LIN {X 0,Y 520.73,Z 981.897,A -85,B 0,C 180,E1 23653.264,E2 23653.264} C_VEL
LIN {X 0,Y 521.246,Z 970.847,A -85,B 0,C 180,E1 23650.972,E2 23650.972} C_VEL
LIN {X 0,Y 521.946,Z 957.782,A -85,B 0,C 180,E1 23648.66,E2 23648.66} C_VEL
LIN {X 0,Y 522.858,Z 943.401,A -85,B 0,C 180,E1 23646.447,E2 23646.447} C_VEL
LIN {X 0,Y 523.895,Z 928.064,A -85,B 0,C 180,E1 23644.403,E2 23644.403} C_VEL
LIN {X 0,Y 525.181,Z 910.158,A -85,B 0,C 180,E1 23642.324,E2 23642.324} C_VEL
LIN {X 0,Y 526.584,Z 891.948,A -85,B 0,C 180,E1 23640.484,E2 23640.484} C_VEL
LIN {X 0,Y 527.978,Z 872.899,A -85,B 0,C 180,E1 23638.832,E2 23638.832} C_VEL
LIN {X 0,Y 529.539,Z 851.797,A -85,B 0,C 180,E1 23637.256,E2 23637.256} C_VEL
LIN {X 0,Y 530.892,Z 831.885,A -85,B 0,C 180,E1 23635.993,E2 23635.993} C_VEL
LIN {X 0,Y 532.275,Z 810.339,A -85,B 0,C 180,E1 23634.853,E2 23634.853} C_VEL
LIN {X 0,Y 533.339,Z 791.087,A -85,B 0,C 180,E1 23634.009,E2 23634.009} C_VEL
LIN {X 0,Y 534.431,Z 767.293,A -85,B 0,C 180,E1 23633.183,E2 23633.183} C_VEL
LIN {X 0,Y 535.229,Z 746.117,A -85,B 0,C 180,E1 23632.64,E2 23632.64} C_VEL
LIN {X 0,Y 535.849,Z 714.207,A -85,B 0,C 180,E1 23632.087,E2 23632.087} C_VEL
LIN {X 0,Y 538.701,Z 503.345,A -85,B 0,C 180,E1 23628.756,E2 23628.756} C_VEL
LIN {X 0,Y 539.867,Z 409.94,A -85,B 0,C 180,E1 23627.231,E2 23627.231} C_VEL
LIN {X 0,Y 537.549,Z 399.203,A -85,B 0,C 180,E1 23626.813,E2 23626.813} C_VEL
LIN {X 0,Y 531.853,Z 390.282,A -85,B 0,C 180,E1 23626.056,E2 23626.056} C_VEL
LIN {X 0,Y 523.904,Z 373.802,A -85,B 0,C 180,E1 23623.836,E2 23623.836} C_VEL
LIN {X 0,Y 520.61,Z 366.663,A -85,B 0,C 180,E1 23622.813,E2 23622.813} C_VEL
LIN {X 0,Y 520.571,Z 366.179,A -85,B 0,C 180,E1 23622.24,E2 23622.24} C_VEL
LIN {X 0,Y 520.51,Z 366.186,A -85,B 0,C 180,E1 23619.054,E2 23619.054} C_VEL
LIN {X 0,Y 520.52,Z 366.183,A -85,B 0,C 180,E1 23615.593,E2 23615.593} C_VEL
LIN {X 0,Y 520.555,Z 366.207,A -85,B 0,C 180,E1 23612.274,E2 23612.274} C_VEL
LIN {X 0,Y 520.498,Z 366.201,A -85,B 0,C 180,E1 23608.952,E2 23608.952} C_VEL
LIN {X 0,Y 520.559,Z 366.202,A -85,B 0,C 180,E1 23605.727,E2 23605.727} C_VEL
LIN {X 0,Y 520.51,Z 366.204,A -85,B 0,C 180,E1 23602.474,E2 23602.474} C_VEL
LIN {X 0,Y 520.513,Z 366.208,A -85,B 0,C 180,E1 23598.943,E2 23598.943} C_VEL
LIN {X 0,Y 520.58,Z 366.205,A -85,B 0,C 180,E1 23595.598,E2 23595.598} C_VEL
LIN {X 0,Y 520.514,Z 366.207,A -85,B 0,C 180,E1 23592.311,E2 23592.311} C_VEL
LIN {X 0,Y 520.532,Z 366.203,A -85,B 0,C 180,E1 23588.839,E2 23588.839} C_VEL
LIN {X 0,Y 520.554,Z 366.207,A -85,B 0,C 180,E1 23585.621,E2 23585.621} C_VEL
LIN {X 0,Y 520.521,Z 366.205,A -85,B 0,C 180,E1 23582.311,E2 23582.311} C_VEL
LIN {X 0,Y 520.584,Z 366.201,A -85,B 0,C 180,E1 23579.009,E2 23579.009} C_VEL
LIN {X 0,Y 520.532,Z 366.206,A -85,B 0,C 180,E1 23575.703,E2 23575.703} C_VEL
LIN {X 0,Y 520.532,Z 366.204,A -85,B 0,C 180,E1 23572.161,E2 23572.161} C_VEL
LIN {X 0,Y 520.589,Z 366.202,A -85,B 0,C 180,E1 23568.814,E2 23568.814} C_VEL
LIN {X 0,Y 520.538,Z 366.205,A -85,B 0,C 180,E1 23565.426,E2 23565.426} C_VEL
LIN {X 0,Y 520.543,Z 366.203,A -85,B 0,C 180,E1 23561.87,E2 23561.87} C_VEL
LIN {X 0,Y 520.59,Z 366.202,A -85,B 0,C 180,E1 23558.479,E2 23558.479} C_VEL
LIN {X 0,Y 520.546,Z 366.202,A -85,B 0,C 180,E1 23555.124,E2 23555.124} C_VEL
LIN {X 0,Y 520.547,Z 366.202,A -85,B 0,C 180,E1 23551.552,E2 23551.552} C_VEL
LIN {X 0,Y 520.589,Z 366.203,A -85,B 0,C 180,E1 23548.247,E2 23548.247} C_VEL
LIN {X 0,Y 520.553,Z 366.202,A -85,B 0,C 180,E1 23544.814,E2 23544.814} C_VEL
LIN {X 0,Y 520.553,Z 366.201,A -85,B 0,C 180,E1 23541.238,E2 23541.238} C_VEL
LIN {X 0,Y 520.585,Z 366.201,A -85,B 0,C 180,E1 23537.841,E2 23537.841} C_VEL
LIN {X 0,Y 520.585,Z 366.201,A -85,B 0,C 180,E1 23537.823,E2 23537.823} C_VEL
LIN {X 0,Y 519.591,Z 366.322,A -85,B 0,C 180,E1 23536.975,E2 23536.975} C_VEL
LIN {X 0,Y 513.168,Z 367.13,A -85,B 0,C 180,E1 23534.593,E2 23534.593} C_VEL
LIN {X 0,Y 512.647,Z 367.188,A -85,B 0,C 180,E1 23533.972,E2 23533.972} C_VEL
LIN {X 0,Y 512.621,Z 367.193,A -85,B 0,C 180,E1 23530.475,E2 23530.475} C_VEL
LIN {X 0,Y 512.626,Z 367.185,A -85,B 0,C 180,E1 23526.899,E2 23526.899} C_VEL
LIN {X 0,Y 512.645,Z 367.191,A -85,B 0,C 180,E1 23523.408,E2 23523.408} C_VEL
LIN {X 0,Y 512.637,Z 367.17,A -85,B 0,C 180,E1 23519.95,E2 23519.95} C_VEL
LIN {X 0,Y 512.626,Z 367.179,A -85,B 0,C 180,E1 23516.457,E2 23516.457} C_VEL
LIN {X 0,Y 512.645,Z 367.187,A -85,B 0,C 180,E1 23512.955,E2 23512.955} C_VEL
LIN {X 0,Y 512.643,Z 367.194,A -85,B 0,C 180,E1 23509.36,E2 23509.36} C_VEL
LIN {X 0,Y 512.631,Z 367.191,A -85,B 0,C 180,E1 23505.843,E2 23505.843} C_VEL
LIN {X 0,Y 512.66,Z 367.389,A -85,B 0,C 180,E1 23504.02,E2 23504.02} C_VEL
LIN {X 0,Y 513.085,Z 368.995,A -85,B 0,C 180,E1 23503.8,E2 23503.8} C_VEL
LIN {X 0,Y 515.161,Z 372.041,A -85,B 0,C 180,E1 23503.498,E2 23503.498} C_VEL
LIN {X 0,Y 516.442,Z 373.536,A -85,B 0,C 180,E1 23503.323,E2 23503.323} C_VEL
LIN {X 0,Y 519.237,Z 377.526,A -85,B 0,C 180,E1 23502.931,E2 23502.931} C_VEL
LIN {X 0,Y 533.14,Z 397.674,A -85,B 0,C 180,E1 23501.079,E2 23501.079} C_VEL
LIN {X 0,Y 533.875,Z 399.243,A -85,B 0,C 180,E1 23500.977,E2 23500.977} C_VEL
LIN {X 0,Y 530.518,Z 616.49,A -85,B 0,C 180,E1 23497.472,E2 23497.472} C_VEL
LIN {X 0,Y 529.04,Z 711.114,A -85,B 0,C 180,E1 23495.95,E2 23495.95} C_VEL
LIN {X 0,Y 528.192,Z 734.087,A -85,B 0,C 180,E1 23495.394,E2 23495.394} C_VEL
LIN {X 0,Y 527.01,Z 757.206,A -85,B 0,C 180,E1 23494.622,E2 23494.622} C_VEL
LIN {X 0,Y 525.757,Z 778.526,A -85,B 0,C 180,E1 23493.704,E2 23493.704} C_VEL
LIN {X 0,Y 524.273,Z 800.117,A -85,B 0,C 180,E1 23492.566,E2 23492.566} C_VEL
LIN {X 0,Y 522.634,Z 821.582,A -85,B 0,C 180,E1 23491.203,E2 23491.203} C_VEL
LIN {X 0,Y 520.941,Z 842.796,A -85,B 0,C 180,E1 23489.604,E2 23489.604} C_VEL
LIN {X 0,Y 519.293,Z 862.614,A -85,B 0,C 180,E1 23487.854,E2 23487.854} C_VEL
LIN {X 0,Y 517.703,Z 881.638,A -85,B 0,C 180,E1 23485.899,E2 23485.899} C_VEL
LIN {X 0,Y 516.28,Z 899.477,A -85,B 0,C 180,E1 23483.771,E2 23483.771} C_VEL
LIN {X 0,Y 515.054,Z 915.866,A -85,B 0,C 180,E1 23481.513,E2 23481.513} C_VEL
LIN {X 0,Y 514.029,Z 930.817,A -85,B 0,C 180,E1 23479.122,E2 23479.122} C_VEL
LIN {X 0,Y 513.257,Z 943.731,A -85,B 0,C 180,E1 23476.708,E2 23476.708} C_VEL
LIN {X 0,Y 512.698,Z 955.351,A -85,B 0,C 180,E1 23474.153,E2 23474.153} C_VEL
LIN {X 0,Y 512.335,Z 964.756,A -85,B 0,C 180,E1 23471.685,E2 23471.685} C_VEL
LIN {X 0,Y 512.081,Z 972.865,A -85,B 0,C 180,E1 23469.062,E2 23469.062} C_VEL
LIN {X 0,Y 511.958,Z 978.812,A -85,B 0,C 180,E1 23466.624,E2 23466.624} C_VEL
LIN {X 0,Y 511.906,Z 983.455,A -85,B 0,C 180,E1 23464.052,E2 23464.052} C_VEL
LIN {X 0,Y 511.912,Z 986.435,A -85,B 0,C 180,E1 23461.515,E2 23461.515} C_VEL
LIN {X 0,Y 511.913,Z 987.823,A -85,B 0,C 180,E1 23458.958,E2 23458.958} C_VEL
LIN {X 0,Y 511.896,Z 987.72,A -85,B 0,C 180,E1 23456.441,E2 23456.441} C_VEL
LIN {X 0,Y 511.906,Z 986.03,A -85,B 0,C 180,E1 23453.963,E2 23453.963} C_VEL
LIN {X 0,Y 511.935,Z 982.848,A -85,B 0,C 180,E1 23451.46,E2 23451.46} C_VEL
LIN {X 0,Y 511.996,Z 977.811,A -85,B 0,C 180,E1 23448.842,E2 23448.842} C_VEL
LIN {X 0,Y 512.139,Z 971.275,A -85,B 0,C 180,E1 23446.279,E2 23446.279} C_VEL
LIN {X 0,Y 512.394,Z 962.857,A -85,B 0,C 180,E1 23443.692,E2 23443.692} C_VEL
LIN {X 0,Y 512.805,Z 952.916,A -85,B 0,C 180,E1 23441.18,E2 23441.18} C_VEL
LIN {X 0,Y 513.371,Z 941.853,A -85,B 0,C 180,E1 23438.824,E2 23438.824} C_VEL
LIN {X 0,Y 514.186,Z 928.411,A -85,B 0,C 180,E1 23436.377,E2 23436.377} C_VEL
LIN {X 0,Y 515.229,Z 913.47,A -85,B 0,C 180,E1 23434.039,E2 23434.039} C_VEL
LIN {X 0,Y 516.43,Z 897.683,A -85,B 0,C 180,E1 23431.908,E2 23431.908} C_VEL
LIN {X 0,Y 517.869,Z 879.852,A -85,B 0,C 180,E1 23429.813,E2 23429.813} C_VEL
LIN {X 0,Y 519.433,Z 860.877,A -85,B 0,C 180,E1 23427.889,E2 23427.889} C_VEL
LIN {X 0,Y 521.061,Z 841.376,A -85,B 0,C 180,E1 23426.19,E2 23426.19} C_VEL
LIN {X 0,Y 522.698,Z 820.709,A -85,B 0,C 180,E1 23424.646,E2 23424.646} C_VEL
LIN {X 0,Y 524.319,Z 799.507,A -85,B 0,C 180,E1 23423.31,E2 23423.31} C_VEL
LIN {X 0,Y 525.799,Z 777.669,A -85,B 0,C 180,E1 23422.166,E2 23422.166} C_VEL
LIN {X 0,Y 527.132,Z 755.086,A -85,B 0,C 180,E1 23421.208,E2 23421.208} C_VEL
LIN {X 0,Y 528.255,Z 732.659,A -85,B 0,C 180,E1 23420.476,E2 23420.476} C_VEL
LIN {X 0,Y 529.11,Z 708.703,A -85,B 0,C 180,E1 23419.911,E2 23419.911} C_VEL
LIN {X 0,Y 532.323,Z 496.573,A -85,B 0,C 180,E1 23416.517,E2 23416.517} C_VEL
LIN {X 0,Y 533.766,Z 398.714,A -85,B 0,C 180,E1 23414.912,E2 23414.912} C_VEL
LIN {X 0,Y 524.776,Z 385.521,A -85,B 0,C 180,E1 23413.728,E2 23413.728} C_VEL
LIN {X 0,Y 518.853,Z 377.145,A -85,B 0,C 180,E1 23412.917,E2 23412.917} C_VEL
LIN {X 0,Y 516.233,Z 373.104,A -85,B 0,C 180,E1 23412.543,E2 23412.543} C_VEL
LIN {X 0,Y 513.441,Z 369.806,A -85,B 0,C 180,E1 23412.152,E2 23412.152} C_VEL
LIN {X 0,Y 512.773,Z 367.944,A -85,B 0,C 180,E1 23411.986,E2 23411.986} C_VEL
LIN {X 0,Y 512.643,Z 367.214,A -85,B 0,C 180,E1 23411.704,E2 23411.704} C_VEL
LIN {X 0,Y 512.646,Z 367.188,A -85,B 0,C 180,E1 23408.186,E2 23408.186} C_VEL
LIN {X 0,Y 512.635,Z 367.191,A -85,B 0,C 180,E1 23404.667,E2 23404.667} C_VEL
LIN {X 0,Y 512.644,Z 367.19,A -85,B 0,C 180,E1 23401.118,E2 23401.118} C_VEL
LIN {X 0,Y 512.626,Z 367.189,A -85,B 0,C 180,E1 23397.653,E2 23397.653} C_VEL
LIN {X 0,Y 512.647,Z 367.189,A -85,B 0,C 180,E1 23394.179,E2 23394.179} C_VEL
LIN {X 0,Y 512.644,Z 367.19,A -85,B 0,C 180,E1 23390.684,E2 23390.684} C_VEL
LIN {X 0,Y 512.611,Z 367.193,A -85,B 0,C 180,E1 23387.233,E2 23387.233} C_VEL
LIN {X 0,Y 512.634,Z 367.194,A -85,B 0,C 180,E1 23383.805,E2 23383.805} C_VEL
LIN {X 0,Y 512.64,Z 367.19,A -85,B 0,C 180,E1 23380.399,E2 23380.399} C_VEL
LIN {X 0,Y 512.595,Z 367.194,A -85,B 0,C 180,E1 23377.027,E2 23377.027} C_VEL
LIN {X 0,Y 512.622,Z 367.196,A -85,B 0,C 180,E1 23373.596,E2 23373.596} C_VEL
LIN {X 0,Y 512.612,Z 367.188,A -85,B 0,C 180,E1 23370.302,E2 23370.302} C_VEL
LIN {X 0,Y 512.577,Z 367.199,A -85,B 0,C 180,E1 23366.895,E2 23366.895} C_VEL
LIN {X 0,Y 512.627,Z 367.19,A -85,B 0,C 180,E1 23363.635,E2 23363.635} C_VEL
LIN {X 0,Y 512.571,Z 367.201,A -85,B 0,C 180,E1 23360.367,E2 23360.367} C_VEL
LIN {X 0,Y 512.632,Z 367.443,A -85,B 0,C 180,E1 23358,E2 23358} C_VEL
LIN {X 0,Y 514.232,Z 371.128,A -85,B 0,C 180,E1 23357.419,E2 23357.419} C_VEL
LIN {X 0,Y 520.729,Z 384.727,A -85,B 0,C 180,E1 23355.506,E2 23355.506} C_VEL
LIN {X 0,Y 523.482,Z 390.317,A -85,B 0,C 180,E1 23354.801,E2 23354.801} C_VEL
LIN {X 0,Y 532.464,Z 404.495,A -85,B 0,C 180,E1 23353.595,E2 23353.595} C_VEL
LIN {X 0,Y 534.046,Z 413.53,A -85,B 0,C 180,E1 23353.27,E2 23353.27} C_VEL
LIN {X 0,Y 530.909,Z 619.639,A -85,B 0,C 180,E1 23349.945,E2 23349.945} C_VEL
LIN {X 0,Y 529.047,Z 740.58,A -85,B 0,C 180,E1 23348.004,E2 23348.004} C_VEL
LIN {X 0,Y 528.186,Z 763.422,A -85,B 0,C 180,E1 23347.452,E2 23347.452} C_VEL
LIN {X 0,Y 527.177,Z 784.197,A -85,B 0,C 180,E1 23346.778,E2 23346.778} C_VEL
LIN {X 0,Y 525.863,Z 806.347,A -85,B 0,C 180,E1 23345.849,E2 23345.849} C_VEL
LIN {X 0,Y 524.539,Z 826.543,A -85,B 0,C 180,E1 23344.815,E2 23344.815} C_VEL
LIN {X 0,Y 522.894,Z 848.108,A -85,B 0,C 180,E1 23343.483,E2 23343.483} C_VEL
LIN {X 0,Y 521.358,Z 867.972,A -85,B 0,C 180,E1 23342.042,E2 23342.042} C_VEL
LIN {X 0,Y 519.726,Z 887.247,A -85,B 0,C 180,E1 23340.398,E2 23340.398} C_VEL
LIN {X 0,Y 518.114,Z 906.768,A -85,B 0,C 180,E1 23338.47,E2 23338.47} C_VEL
LIN {X 0,Y 516.729,Z 923.641,A -85,B 0,C 180,E1 23336.552,E2 23336.552} C_VEL
LIN {X 0,Y 515.543,Z 939.129,A -85,B 0,C 180,E1 23334.524,E2 23334.524} C_VEL
LIN {X 0,Y 514.478,Z 954.207,A -85,B 0,C 180,E1 23332.272,E2 23332.272} C_VEL
LIN {X 0,Y 513.632,Z 967.078,A -85,B 0,C 180,E1 23330.038,E2 23330.038} C_VEL
LIN {X 0,Y 512.948,Z 979.795,A -85,B 0,C 180,E1 23327.471,E2 23327.471} C_VEL
LIN {X 0,Y 512.523,Z 989.52,A -85,B 0,C 180,E1 23325.156,E2 23325.156} C_VEL
LIN {X 0,Y 512.205,Z 998.523,A -85,B 0,C 180,E1 23322.572,E2 23322.572} C_VEL
LIN {X 0,Y 512.02,Z 1005.466,A -85,B 0,C 180,E1 23320.125,E2 23320.125} C_VEL
LIN {X 0,Y 511.944,Z 1010.836,A -85,B 0,C 180,E1 23317.635,E2 23317.635} C_VEL
LIN {X 0,Y 511.916,Z 1014.592,A -85,B 0,C 180,E1 23315.27,E2 23315.27} C_VEL
LIN {X 0,Y 511.903,Z 1017.053,A -85,B 0,C 180,E1 23312.69,E2 23312.69} C_VEL
LIN {X 0,Y 511.887,Z 1017.916,A -85,B 0,C 180,E1 23310.451,E2 23310.451} C_VEL
LIN {X 0,Y 511.914,Z 1017.394,A -85,B 0,C 180,E1 23307.876,E2 23307.876} C_VEL
LIN {X 0,Y 511.905,Z 1015.505,A -85,B 0,C 180,E1 23305.522,E2 23305.522} C_VEL
LIN {X 0,Y 511.913,Z 1011.88,A -85,B 0,C 180,E1 23302.935,E2 23302.935} C_VEL
LIN {X 0,Y 511.996,Z 1007.326,A -85,B 0,C 180,E1 23300.675,E2 23300.675} C_VEL
LIN {X 0,Y 512.153,Z 1000.479,A -85,B 0,C 180,E1 23298.06,E2 23298.06} C_VEL
LIN {X 0,Y 512.376,Z 992.946,A -85,B 0,C 180,E1 23295.77,E2 23295.77} C_VEL
LIN {X 0,Y 512.8,Z 982.809,A -85,B 0,C 180,E1 23293.205,E2 23293.205} C_VEL
LIN {X 0,Y 513.349,Z 972.01,A -85,B 0,C 180,E1 23290.904,E2 23290.904} C_VEL
LIN {X 0,Y 514.167,Z 958.481,A -85,B 0,C 180,E1 23288.44,E2 23288.44} C_VEL
LIN {X 0,Y 515.173,Z 944.243,A -85,B 0,C 180,E1 23286.195,E2 23286.195} C_VEL
LIN {X 0,Y 516.359,Z 928.443,A -85,B 0,C 180,E1 23284.052,E2 23284.052} C_VEL
LIN {X 0,Y 517.829,Z 910.156,A -85,B 0,C 180,E1 23281.897,E2 23281.897} C_VEL
LIN {X 0,Y 519.361,Z 891.964,A -85,B 0,C 180,E1 23280.034,E2 23280.034} C_VEL
LIN {X 0,Y 520.943,Z 872.64,A -85,B 0,C 180,E1 23278.341,E2 23278.341} C_VEL
LIN {X 0,Y 522.622,Z 851.799,A -85,B 0,C 180,E1 23276.767,E2 23276.767} C_VEL
LIN {X 0,Y 524.127,Z 831.882,A -85,B 0,C 180,E1 23275.493,E2 23275.493} C_VEL
LIN {X 0,Y 525.674,Z 809.636,A -85,B 0,C 180,E1 23274.308,E2 23274.308} C_VEL
LIN {X 0,Y 526.874,Z 789.605,A -85,B 0,C 180,E1 23273.429,E2 23273.429} C_VEL
LIN {X 0,Y 528.036,Z 766.565,A -85,B 0,C 180,E1 23272.638,E2 23272.638} C_VEL
LIN {X 0,Y 528.897,Z 745.467,A -85,B 0,C 180,E1 23272.097,E2 23272.097} C_VEL
LIN {X 0,Y 529.568,Z 712.31,A -85,B 0,C 180,E1 23271.524,E2 23271.524} C_VEL
LIN {X 0,Y 532.699,Z 501.745,A -85,B 0,C 180,E1 23268.162,E2 23268.162} C_VEL
LIN {X 0,Y 533.925,Z 411.726,A -85,B 0,C 180,E1 23266.679,E2 23266.679} C_VEL
LIN {X 0,Y 532.155,Z 403.642,A -85,B 0,C 180,E1 23266.352,E2 23266.352} C_VEL
LIN {X 0,Y 523.286,Z 389.924,A -85,B 0,C 180,E1 23265.143,E2 23265.143} C_VEL
LIN {X 0,Y 516.279,Z 375.3,A -85,B 0,C 180,E1 23263.11,E2 23263.11} C_VEL
LIN {X 0,Y 512.667,Z 367.602,A -85,B 0,C 180,E1 23261.958,E2 23261.958} C_VEL
LIN {X 0,Y 512.576,Z 367.194,A -85,B 0,C 180,E1 23261.099,E2 23261.099} C_VEL
LIN {X 0,Y 512.584,Z 367.2,A -85,B 0,C 180,E1 23257.628,E2 23257.628} C_VEL
LIN {X 0,Y 512.615,Z 367.169,A -85,B 0,C 180,E1 23254.311,E2 23254.311} C_VEL
LIN {X 0,Y 512.563,Z 367.18,A -85,B 0,C 180,E1 23250.996,E2 23250.996} C_VEL
LIN {X 0,Y 512.606,Z 367.198,A -85,B 0,C 180,E1 23247.66,E2 23247.66} C_VEL
LIN {X 0,Y 512.579,Z 367.198,A -85,B 0,C 180,E1 23244.375,E2 23244.375} C_VEL
LIN {X 0,Y 512.568,Z 367.196,A -85,B 0,C 180,E1 23240.914,E2 23240.914} C_VEL
LIN {X 0,Y 512.634,Z 367.189,A -85,B 0,C 180,E1 23237.596,E2 23237.596} C_VEL
LIN {X 0,Y 512.573,Z 367.193,A -85,B 0,C 180,E1 23234.343,E2 23234.343} C_VEL
LIN {X 0,Y 512.592,Z 367.192,A -85,B 0,C 180,E1 23230.906,E2 23230.906} C_VEL
LIN {X 0,Y 512.62,Z 367.189,A -85,B 0,C 180,E1 23227.621,E2 23227.621} C_VEL
LIN {X 0,Y 512.579,Z 367.189,A -85,B 0,C 180,E1 23224.251,E2 23224.251} C_VEL
LIN {X 0,Y 512.628,Z 367.19,A -85,B 0,C 180,E1 23220.894,E2 23220.894} C_VEL
LIN {X 0,Y 512.598,Z 367.191,A -85,B 0,C 180,E1 23217.652,E2 23217.652} C_VEL
LIN {X 0,Y 512.591,Z 367.187,A -85,B 0,C 180,E1 23214.178,E2 23214.178} C_VEL
LIN {X 0,Y 512.648,Z 367.186,A -85,B 0,C 180,E1 23210.797,E2 23210.797} C_VEL
LIN {X 0,Y 512.605,Z 367.193,A -85,B 0,C 180,E1 23207.381,E2 23207.381} C_VEL
LIN {X 0,Y 512.601,Z 367.188,A -85,B 0,C 180,E1 23203.92,E2 23203.92} C_VEL
LIN {X 0,Y 512.65,Z 367.184,A -85,B 0,C 180,E1 23200.517,E2 23200.517} C_VEL
LIN {X 0,Y 512.608,Z 367.194,A -85,B 0,C 180,E1 23197.16,E2 23197.16} C_VEL
LIN {X 0,Y 512.607,Z 367.189,A -85,B 0,C 180,E1 23193.594,E2 23193.594} C_VEL
LIN {X 0,Y 512.651,Z 367.184,A -85,B 0,C 180,E1 23190.175,E2 23190.175} C_VEL
LIN {X 0,Y 512.621,Z 367.194,A -85,B 0,C 180,E1 23186.764,E2 23186.764} C_VEL
LIN {X 0,Y 512.61,Z 367.19,A -85,B 0,C 180,E1 23183.215,E2 23183.215} C_VEL
LIN {X 0,Y 512.649,Z 367.182,A -85,B 0,C 180,E1 23179.791,E2 23179.791} C_VEL
LIN {X 0,Y 512.635,Z 367.189,A -85,B 0,C 180,E1 23176.334,E2 23176.334} C_VEL
LIN {X 0,Y 512.647,Z 367.188,A -85,B 0,C 180,E1 23173.972,E2 23173.972} C_VEL
LIN {X 0,Y 511.668,Z 367.306,A -85,B 0,C 180,E1 23173.111,E2 23173.111} C_VEL
LIN {X 0,Y 505.23,Z 368.113,A -85,B 0,C 180,E1 23170.692,E2 23170.692} C_VEL
LIN {X 0,Y 504.706,Z 368.176,A -85,B 0,C 180,E1 23170.061,E2 23170.061} C_VEL
LIN {X 0,Y 504.68,Z 368.176,A -85,B 0,C 180,E1 23166.602,E2 23166.602} C_VEL
LIN {X 0,Y 504.706,Z 368.178,A -85,B 0,C 180,E1 23163.071,E2 23163.071} C_VEL
LIN {X 0,Y 504.704,Z 368.162,A -85,B 0,C 180,E1 23159.552,E2 23159.552} C_VEL
LIN {X 0,Y 504.688,Z 368.161,A -85,B 0,C 180,E1 23156.088,E2 23156.088} C_VEL
LIN {X 0,Y 504.693,Z 368.173,A -85,B 0,C 180,E1 23152.476,E2 23152.476} C_VEL
LIN {X 0,Y 504.702,Z 368.179,A -85,B 0,C 180,E1 23148.956,E2 23148.956} C_VEL
LIN {X 0,Y 504.707,Z 368.178,A -85,B 0,C 180,E1 23145.391,E2 23145.391} C_VEL
LIN {X 0,Y 504.748,Z 368.504,A -85,B 0,C 180,E1 23144.919,E2 23144.919} C_VEL
LIN {X 0,Y 505.276,Z 370.293,A -85,B 0,C 180,E1 23144.696,E2 23144.696} C_VEL
LIN {X 0,Y 507.471,Z 373.261,A -85,B 0,C 180,E1 23144.371,E2 23144.371} C_VEL
LIN {X 0,Y 508.566,Z 374.536,A -85,B 0,C 180,E1 23144.215,E2 23144.215} C_VEL
LIN {X 0,Y 511.339,Z 378.515,A -85,B 0,C 180,E1 23143.809,E2 23143.809} C_VEL
LIN {X 0,Y 523.571,Z 395.963,A -85,B 0,C 180,E1 23142.105,E2 23142.105} C_VEL
LIN {X 0,Y 527.971,Z 402.706,A -85,B 0,C 180,E1 23141.515,E2 23141.515} C_VEL
LIN {X 0,Y 524.271,Z 621.523,A -85,B 0,C 180,E1 23137.95,E2 23137.95} C_VEL
LIN {X 0,Y 522.729,Z 711.176,A -85,B 0,C 180,E1 23136.49,E2 23136.49} C_VEL
LIN {X 0,Y 521.821,Z 734.082,A -85,B 0,C 180,E1 23135.932,E2 23135.932} C_VEL
LIN {X 0,Y 520.552,Z 756.976,A -85,B 0,C 180,E1 23135.163,E2 23135.163} C_VEL
LIN {X 0,Y 519.121,Z 779.272,A -85,B 0,C 180,E1 23134.194,E2 23134.194} C_VEL
LIN {X 0,Y 517.511,Z 800.76,A -85,B 0,C 180,E1 23133.043,E2 23133.043} C_VEL
LIN {X 0,Y 515.779,Z 821.379,A -85,B 0,C 180,E1 23131.719,E2 23131.719} C_VEL
LIN {X 0,Y 513.93,Z 842.647,A -85,B 0,C 180,E1 23130.1,E2 23130.1} C_VEL
LIN {X 0,Y 512.093,Z 862.604,A -85,B 0,C 180,E1 23128.319,E2 23128.319} C_VEL
LIN {X 0,Y 510.378,Z 881.548,A -85,B 0,C 180,E1 23126.347,E2 23126.347} C_VEL
LIN {X 0,Y 508.831,Z 898.974,A -85,B 0,C 180,E1 23124.246,E2 23124.246} C_VEL
LIN {X 0,Y 507.513,Z 914.669,A -85,B 0,C 180,E1 23122.07,E2 23122.07} C_VEL
LIN {X 0,Y 506.416,Z 929.109,A -85,B 0,C 180,E1 23119.762,E2 23119.762} C_VEL
LIN {X 0,Y 505.489,Z 942.81,A -85,B 0,C 180,E1 23117.198,E2 23117.198} C_VEL
LIN {X 0,Y 504.853,Z 954.246,A -85,B 0,C 180,E1 23114.689,E2 23114.689} C_VEL
LIN {X 0,Y 504.411,Z 964.063,A -85,B 0,C 180,E1 23112.104,E2 23112.104} C_VEL
LIN {X 0,Y 504.13,Z 972.325,A -85,B 0,C 180,E1 23109.446,E2 23109.446} C_VEL
LIN {X 0,Y 503.991,Z 978.303,A -85,B 0,C 180,E1 23106.992,E2 23106.992} C_VEL
LIN {X 0,Y 503.929,Z 983.128,A -85,B 0,C 180,E1 23104.369,E2 23104.369} C_VEL
LIN {X 0,Y 503.912,Z 986.272,A -85,B 0,C 180,E1 23101.761,E2 23101.761} C_VEL
LIN {X 0,Y 503.917,Z 987.805,A -85,B 0,C 180,E1 23099.074,E2 23099.074} C_VEL
LIN {X 0,Y 503.906,Z 987.77,A -85,B 0,C 180,E1 23096.653,E2 23096.653} C_VEL
LIN {X 0,Y 503.908,Z 986.163,A -85,B 0,C 180,E1 23094.03,E2 23094.03} C_VEL
LIN {X 0,Y 503.937,Z 982.944,A -85,B 0,C 180,E1 23091.42,E2 23091.42} C_VEL
LIN {X 0,Y 504.009,Z 977.938,A -85,B 0,C 180,E1 23088.753,E2 23088.753} C_VEL
LIN {X 0,Y 504.163,Z 971.583,A -85,B 0,C 180,E1 23086.198,E2 23086.198} C_VEL
LIN {X 0,Y 504.435,Z 963.388,A -85,B 0,C 180,E1 23083.613,E2 23083.613} C_VEL
LIN {X 0,Y 504.897,Z 953.381,A -85,B 0,C 180,E1 23081.016,E2 23081.016} C_VEL
LIN {X 0,Y 505.551,Z 941.949,A -85,B 0,C 180,E1 23078.536,E2 23078.536} C_VEL
LIN {X 0,Y 506.466,Z 928.453,A -85,B 0,C 180,E1 23076.037,E2 23076.037} C_VEL
LIN {X 0,Y 507.619,Z 913.458,A -85,B 0,C 180,E1 23073.655,E2 23073.655} C_VEL
LIN {X 0,Y 508.974,Z 897.303,A -85,B 0,C 180,E1 23071.446,E2 23071.446} C_VEL
LIN {X 0,Y 510.551,Z 879.8,A -85,B 0,C 180,E1 23069.366,E2 23069.366} C_VEL
LIN {X 0,Y 512.252,Z 860.935,A -85,B 0,C 180,E1 23067.429,E2 23067.429} C_VEL
LIN {X 0,Y 514.044,Z 841.395,A -85,B 0,C 180,E1 23065.706,E2 23065.706} C_VEL
LIN {X 0,Y 515.842,Z 820.666,A -85,B 0,C 180,E1 23064.141,E2 23064.141} C_VEL
LIN {X 0,Y 517.611,Z 799.469,A -85,B 0,C 180,E1 23062.793,E2 23062.793} C_VEL
LIN {X 0,Y 519.208,Z 777.68,A -85,B 0,C 180,E1 23061.641,E2 23061.641} C_VEL
LIN {X 0,Y 520.686,Z 754.91,A -85,B 0,C 180,E1 23060.669,E2 23060.669} C_VEL
LIN {X 0,Y 521.881,Z 732.723,A -85,B 0,C 180,E1 23059.94,E2 23059.94} C_VEL
LIN {X 0,Y 522.803,Z 708.819,A -85,B 0,C 180,E1 23059.371,E2 23059.371} C_VEL
LIN {X 0,Y 526.211,Z 502.36,A -85,B 0,C 180,E1 23056.036,E2 23056.036} C_VEL
LIN {X 0,Y 527.849,Z 402.167,A -85,B 0,C 180,E1 23054.368,E2 23054.368} C_VEL
LIN {X 0,Y 515.031,Z 383.624,A -85,B 0,C 180,E1 23052.616,E2 23052.616} C_VEL
LIN {X 0,Y 510.951,Z 378.14,A -85,B 0,C 180,E1 23052.029,E2 23052.029} C_VEL
LIN {X 0,Y 507.813,Z 373.554,A -85,B 0,C 180,E1 23051.557,E2 23051.557} C_VEL
LIN {X 0,Y 505.45,Z 370.685,A -85,B 0,C 180,E1 23051.207,E2 23051.207} C_VEL
LIN {X 0,Y 504.863,Z 369.085,A -85,B 0,C 180,E1 23051.076,E2 23051.076} C_VEL
LIN {X 0,Y 504.693,Z 368.209,A -85,B 0,C 180,E1 23050.791,E2 23050.791} C_VEL
LIN {X 0,Y 504.711,Z 368.18,A -85,B 0,C 180,E1 23047.284,E2 23047.284} C_VEL
LIN {X 0,Y 504.694,Z 368.181,A -85,B 0,C 180,E1 23043.749,E2 23043.749} C_VEL
LIN {X 0,Y 504.706,Z 368.177,A -85,B 0,C 180,E1 23040.227,E2 23040.227} C_VEL
LIN {X 0,Y 504.705,Z 368.177,A -85,B 0,C 180,E1 23036.707,E2 23036.707} C_VEL
LIN {X 0,Y 504.685,Z 368.178,A -85,B 0,C 180,E1 23033.174,E2 23033.174} C_VEL
LIN {X 0,Y 504.683,Z 368.182,A -85,B 0,C 180,E1 23029.614,E2 23029.614} C_VEL
LIN {X 0,Y 504.713,Z 368.18,A -85,B 0,C 180,E1 23026.103,E2 23026.103} C_VEL
LIN {X 0,Y 504.692,Z 368.18,A -85,B 0,C 180,E1 23022.594,E2 23022.594} C_VEL
LIN {X 0,Y 504.66,Z 368.184,A -85,B 0,C 180,E1 23019.107,E2 23019.107} C_VEL
LIN {X 0,Y 504.687,Z 368.179,A -85,B 0,C 180,E1 23015.665,E2 23015.665} C_VEL
LIN {X 0,Y 504.686,Z 368.181,A -85,B 0,C 180,E1 23012.253,E2 23012.253} C_VEL
LIN {X 0,Y 504.642,Z 368.186,A -85,B 0,C 180,E1 23008.861,E2 23008.861} C_VEL
LIN {X 0,Y 504.674,Z 368.179,A -85,B 0,C 180,E1 23005.485,E2 23005.485} C_VEL
LIN {X 0,Y 504.658,Z 368.188,A -85,B 0,C 180,E1 23002.107,E2 23002.107} C_VEL
LIN {X 0,Y 504.66,Z 368.402,A -85,B 0,C 180,E1 22998.895,E2 22998.895} C_VEL
LIN {X 0,Y 506.098,Z 371.902,A -85,B 0,C 180,E1 22998.315,E2 22998.315} C_VEL
LIN {X 0,Y 511.144,Z 382.049,A -85,B 0,C 180,E1 22996.793,E2 22996.793} C_VEL
LIN {X 0,Y 514.801,Z 389.529,A -85,B 0,C 180,E1 22995.774,E2 22995.774} C_VEL
LIN {X 0,Y 527.065,Z 408.685,A -85,B 0,C 180,E1 22994.07,E2 22994.07} C_VEL
LIN {X 0,Y 528.155,Z 415.317,A -85,B 0,C 180,E1 22993.833,E2 22993.833} C_VEL
LIN {X 0,Y 524.723,Z 622.728,A -85,B 0,C 180,E1 22990.457,E2 22990.457} C_VEL
LIN {X 0,Y 522.741,Z 740.58,A -85,B 0,C 180,E1 22988.546,E2 22988.546} C_VEL
LIN {X 0,Y 521.82,Z 763.29,A -85,B 0,C 180,E1 22987.994,E2 22987.994} C_VEL
LIN {X 0,Y 520.774,Z 783.33,A -85,B 0,C 180,E1 22987.341,E2 22987.341} C_VEL
LIN {X 0,Y 519.282,Z 806.344,A -85,B 0,C 180,E1 22986.375,E2 22986.375} C_VEL
LIN {X 0,Y 517.769,Z 827.665,A -85,B 0,C 180,E1 22985.27,E2 22985.27} C_VEL
LIN {X 0,Y 516.052,Z 848.22,A -85,B 0,C 180,E1 22983.978,E2 22983.978} C_VEL
LIN {X 0,Y 514.337,Z 868.231,A -85,B 0,C 180,E1 22982.51,E2 22982.51} C_VEL
LIN {X 0,Y 512.591,Z 887.244,A -85,B 0,C 180,E1 22980.866,E2 22980.866} C_VEL
LIN {X 0,Y 510.803,Z 906.767,A -85,B 0,C 180,E1 22978.915,E2 22978.915} C_VEL
LIN {X 0,Y 509.335,Z 923.134,A -85,B 0,C 180,E1 22977.032,E2 22977.032} C_VEL
LIN {X 0,Y 507.971,Z 939.128,A -85,B 0,C 180,E1 22974.914,E2 22974.914} C_VEL
LIN {X 0,Y 506.777,Z 954.209,A -85,B 0,C 180,E1 22972.629,E2 22972.629} C_VEL
LIN {X 0,Y 505.847,Z 967.076,A -85,B 0,C 180,E1 22970.36,E2 22970.36} C_VEL
LIN {X 0,Y 505.089,Z 979.615,A -85,B 0,C 180,E1 22967.793,E2 22967.793} C_VEL
LIN {X 0,Y 504.599,Z 989.518,A -85,B 0,C 180,E1 22965.4,E2 22965.4} C_VEL
LIN {X 0,Y 504.253,Z 998.339,A -85,B 0,C 180,E1 22962.834,E2 22962.834} C_VEL
LIN {X 0,Y 504.057,Z 1005.162,A -85,B 0,C 180,E1 22960.402,E2 22960.402} C_VEL
LIN {X 0,Y 503.97,Z 1010.63,A -85,B 0,C 180,E1 22957.871,E2 22957.871} C_VEL
LIN {X 0,Y 503.912,Z 1014.433,A -85,B 0,C 180,E1 22955.468,E2 22955.468} C_VEL
LIN {X 0,Y 503.895,Z 1016.985,A -85,B 0,C 180,E1 22952.846,E2 22952.846} C_VEL
LIN {X 0,Y 503.884,Z 1017.894,A -85,B 0,C 180,E1 22950.571,E2 22950.571} C_VEL
LIN {X 0,Y 503.914,Z 1017.394,A -85,B 0,C 180,E1 22947.843,E2 22947.843} C_VEL
LIN {X 0,Y 503.905,Z 1015.505,A -85,B 0,C 180,E1 22945.451,E2 22945.451} C_VEL
LIN {X 0,Y 503.919,Z 1011.807,A -85,B 0,C 180,E1 22942.782,E2 22942.782} C_VEL
LIN {X 0,Y 504,Z 1007.326,A -85,B 0,C 180,E1 22940.526,E2 22940.526} C_VEL
LIN {X 0,Y 504.182,Z 1000.479,A -85,B 0,C 180,E1 22937.869,E2 22937.869} C_VEL
LIN {X 0,Y 504.445,Z 992.948,A -85,B 0,C 180,E1 22935.541,E2 22935.541} C_VEL
LIN {X 0,Y 504.912,Z 982.923,A -85,B 0,C 180,E1 22932.961,E2 22932.961} C_VEL
LIN {X 0,Y 505.538,Z 972.012,A -85,B 0,C 180,E1 22930.597,E2 22930.597} C_VEL
LIN {X 0,Y 506.453,Z 958.479,A -85,B 0,C 180,E1 22928.095,E2 22928.095} C_VEL
LIN {X 0,Y 507.573,Z 944.064,A -85,B 0,C 180,E1 22925.79,E2 22925.79} C_VEL
LIN {X 0,Y 508.879,Z 928.364,A -85,B 0,C 180,E1 22923.631,E2 22923.631} C_VEL
LIN {X 0,Y 510.5,Z 910.155,A -85,B 0,C 180,E1 22921.456,E2 22921.456} C_VEL
LIN {X 0,Y 512.149,Z 892.226,A -85,B 0,C 180,E1 22919.594,E2 22919.594} C_VEL
LIN {X 0,Y 513.853,Z 873.371,A -85,B 0,C 180,E1 22917.918,E2 22917.918} C_VEL
LIN {X 0,Y 515.615,Z 853.583,A -85,B 0,C 180,E1 22916.389,E2 22916.389} C_VEL
LIN {X 0,Y 517.227,Z 833.888,A -85,B 0,C 180,E1 22915.101,E2 22915.101} C_VEL
LIN {X 0,Y 518.955,Z 811.617,A -85,B 0,C 180,E1 22913.879,E2 22913.879} C_VEL
LIN {X 0,Y 520.29,Z 791.081,A -85,B 0,C 180,E1 22912.959,E2 22912.959} C_VEL
LIN {X 0,Y 521.625,Z 767.163,A -85,B 0,C 180,E1 22912.119,E2 22912.119} C_VEL
LIN {X 0,Y 522.527,Z 746.603,A -85,B 0,C 180,E1 22911.582,E2 22911.582} C_VEL
LIN {X 0,Y 523.264,Z 715.237,A -85,B 0,C 180,E1 22911.023,E2 22911.023} C_VEL
LIN {X 0,Y 526.658,Z 504.557,A -85,B 0,C 180,E1 22907.63,E2 22907.63} C_VEL
LIN {X 0,Y 528.058,Z 413.604,A -85,B 0,C 180,E1 22906.118,E2 22906.118} C_VEL
LIN {X 0,Y 526.801,Z 408.028,A -85,B 0,C 180,E1 22905.882,E2 22905.882} C_VEL
LIN {X 0,Y 514.855,Z 389.56,A -85,B 0,C 180,E1 22904.201,E2 22904.201} C_VEL
LIN {X 0,Y 507.975,Z 375.58,A -85,B 0,C 180,E1 22902.159,E2 22902.159} C_VEL
LIN {X 0,Y 506.106,Z 371.905,A -85,B 0,C 180,E1 22901.59,E2 22901.59} C_VEL
LIN {X 0,Y 504.669,Z 368.389,A -85,B 0,C 180,E1 22901.012,E2 22901.012} C_VEL
LIN {X 0,Y 504.667,Z 368.177,A -85,B 0,C 180,E1 22897.892,E2 22897.892} C_VEL
LIN {X 0,Y 504.642,Z 368.157,A -85,B 0,C 180,E1 22894.655,E2 22894.655} C_VEL
LIN {X 0,Y 504.628,Z 368.171,A -85,B 0,C 180,E1 22891.273,E2 22891.273} C_VEL
LIN {X 0,Y 504.698,Z 368.179,A -85,B 0,C 180,E1 22887.934,E2 22887.934} C_VEL
LIN {X 0,Y 504.63,Z 368.187,A -85,B 0,C 180,E1 22884.583,E2 22884.583} C_VEL
LIN {X 0,Y 504.634,Z 368.185,A -85,B 0,C 180,E1 22881.015,E2 22881.015} C_VEL
LIN {X 0,Y 504.695,Z 368.178,A -85,B 0,C 180,E1 22877.644,E2 22877.644} C_VEL
LIN {X 0,Y 504.634,Z 368.182,A -85,B 0,C 180,E1 22874.339,E2 22874.339} C_VEL
LIN {X 0,Y 504.649,Z 368.181,A -85,B 0,C 180,E1 22870.849,E2 22870.849} C_VEL
LIN {X 0,Y 504.692,Z 368.177,A -85,B 0,C 180,E1 22867.513,E2 22867.513} C_VEL
LIN {X 0,Y 504.643,Z 368.178,A -85,B 0,C 180,E1 22864.09,E2 22864.09} C_VEL
LIN {X 0,Y 504.659,Z 368.181,A -85,B 0,C 180,E1 22860.567,E2 22860.567} C_VEL
LIN {X 0,Y 504.692,Z 368.177,A -85,B 0,C 180,E1 22857.274,E2 22857.274} C_VEL
LIN {X 0,Y 504.649,Z 368.176,A -85,B 0,C 180,E1 22853.858,E2 22853.858} C_VEL
LIN {X 0,Y 504.678,Z 368.178,A -85,B 0,C 180,E1 22850.42,E2 22850.42} C_VEL
LIN {X 0,Y 504.69,Z 368.177,A -85,B 0,C 180,E1 22847.063,E2 22847.063} C_VEL
LIN {X 0,Y 504.657,Z 368.177,A -85,B 0,C 180,E1 22843.659,E2 22843.659} C_VEL
LIN {X 0,Y 504.691,Z 368.172,A -85,B 0,C 180,E1 22840.198,E2 22840.198} C_VEL
LIN {X 0,Y 504.697,Z 368.177,A -85,B 0,C 180,E1 22836.781,E2 22836.781} C_VEL
LIN {X 0,Y 504.665,Z 368.179,A -85,B 0,C 180,E1 22833.31,E2 22833.31} C_VEL
LIN {X 0,Y 504.701,Z 368.172,A -85,B 0,C 180,E1 22829.919,E2 22829.919} C_VEL
LIN {X 0,Y 504.703,Z 368.177,A -85,B 0,C 180,E1 22826.446,E2 22826.446} C_VEL
LIN {X 0,Y 504.671,Z 368.18,A -85,B 0,C 180,E1 22822.966,E2 22822.966} C_VEL
LIN {X 0,Y 504.694,Z 368.171,A -85,B 0,C 180,E1 22819.473,E2 22819.473} C_VEL
LIN {X 0,Y 504.708,Z 368.176,A -85,B 0,C 180,E1 22815.944,E2 22815.944} C_VEL
LIN {X 0,Y 504.682,Z 368.176,A -85,B 0,C 180,E1 22812.493,E2 22812.493} C_VEL
LIN {X 0,Y 504.706,Z 368.176,A -85,B 0,C 180,E1 22810.061,E2 22810.061} C_VEL
LIN {X 0,Y 503.723,Z 368.301,A -85,B 0,C 180,E1 22809.186,E2 22809.186} C_VEL
LIN {X 0,Y 497.271,Z 369.1,A -85,B 0,C 180,E1 22806.728,E2 22806.728} C_VEL
LIN {X 0,Y 496.757,Z 369.169,A -85,B 0,C 180,E1 22806.087,E2 22806.087} C_VEL
LIN {X 0,Y 496.746,Z 369.17,A -85,B 0,C 180,E1 22802.502,E2 22802.502} C_VEL
LIN {X 0,Y 496.768,Z 369.161,A -85,B 0,C 180,E1 22799.012,E2 22799.012} C_VEL
LIN {X 0,Y 496.764,Z 369.144,A -85,B 0,C 180,E1 22795.509,E2 22795.509} C_VEL
LIN {X 0,Y 496.751,Z 369.151,A -85,B 0,C 180,E1 22791.982,E2 22791.982} C_VEL
LIN {X 0,Y 496.761,Z 369.155,A -85,B 0,C 180,E1 22788.417,E2 22788.417} C_VEL
LIN {X 0,Y 496.774,Z 369.326,A -85,B 0,C 180,E1 22785.942,E2 22785.942} C_VEL
LIN {X 0,Y 497.138,Z 370.8,A -85,B 0,C 180,E1 22785.701,E2 22785.701} C_VEL
LIN {X 0,Y 499.073,Z 373.858,A -85,B 0,C 180,E1 22785.387,E2 22785.387} C_VEL
LIN {X 0,Y 500.705,Z 375.539,A -85,B 0,C 180,E1 22785.148,E2 22785.148} C_VEL
LIN {X 0,Y 503.468,Z 379.538,A -85,B 0,C 180,E1 22784.724,E2 22784.724} C_VEL
LIN {X 0,Y 512.807,Z 392.598,A -85,B 0,C 180,E1 22783.359,E2 22783.359} C_VEL
LIN {X 0,Y 522.12,Z 406.25,A -85,B 0,C 180,E1 22782.064,E2 22782.064} C_VEL
LIN {X 0,Y 518.072,Z 624.59,A -85,B 0,C 180,E1 22778.468,E2 22778.468} C_VEL
LIN {X 0,Y 516.472,Z 711.072,A -85,B 0,C 180,E1 22777.048,E2 22777.048} C_VEL
LIN {X 0,Y 515.503,Z 733.955,A -85,B 0,C 180,E1 22776.487,E2 22776.487} C_VEL
LIN {X 0,Y 514.147,Z 756.737,A -85,B 0,C 180,E1 22775.717,E2 22775.717} C_VEL
LIN {X 0,Y 512.598,Z 778.858,A -85,B 0,C 180,E1 22774.752,E2 22774.752} C_VEL
LIN {X 0,Y 510.908,Z 799.877,A -85,B 0,C 180,E1 22773.621,E2 22773.621} C_VEL
LIN {X 0,Y 508.983,Z 821.162,A -85,B 0,C 180,E1 22772.249,E2 22772.249} C_VEL
LIN {X 0,Y 506.959,Z 842.494,A -85,B 0,C 180,E1 22770.61,E2 22770.61} C_VEL
LIN {X 0,Y 504.951,Z 862.494,A -85,B 0,C 180,E1 22768.806,E2 22768.806} C_VEL
LIN {X 0,Y 503.081,Z 881.462,A -85,B 0,C 180,E1 22766.807,E2 22766.807} C_VEL
LIN {X 0,Y 501.324,Z 899.351,A -85,B 0,C 180,E1 22764.618,E2 22764.618} C_VEL
LIN {X 0,Y 499.817,Z 915.749,A -85,B 0,C 180,E1 22762.295,E2 22762.295} C_VEL
LIN {X 0,Y 498.615,Z 930.155,A -85,B 0,C 180,E1 22759.929,E2 22759.929} C_VEL
LIN {X 0,Y 497.662,Z 943.039,A -85,B 0,C 180,E1 22757.465,E2 22757.465} C_VEL
LIN {X 0,Y 496.963,Z 954.275,A -85,B 0,C 180,E1 22754.955,E2 22754.955} C_VEL
LIN {X 0,Y 496.482,Z 963.793,A -85,B 0,C 180,E1 22752.415,E2 22752.415} C_VEL
LIN {X 0,Y 496.179,Z 972.106,A -85,B 0,C 180,E1 22749.718,E2 22749.718} C_VEL
LIN {X 0,Y 496.007,Z 978.373,A -85,B 0,C 180,E1 22747.107,E2 22747.107} C_VEL
LIN {X 0,Y 495.934,Z 983.178,A -85,B 0,C 180,E1 22744.438,E2 22744.438} C_VEL
LIN {X 0,Y 495.913,Z 986.359,A -85,B 0,C 180,E1 22741.716,E2 22741.716} C_VEL
LIN {X 0,Y 495.917,Z 987.813,A -85,B 0,C 180,E1 22739.059,E2 22739.059} C_VEL
LIN {X 0,Y 495.903,Z 987.762,A -85,B 0,C 180,E1 22736.587,E2 22736.587} C_VEL
LIN {X 0,Y 495.903,Z 986.13,A -85,B 0,C 180,E1 22733.93,E2 22733.93} C_VEL
LIN {X 0,Y 495.939,Z 982.894,A -85,B 0,C 180,E1 22731.282,E2 22731.282} C_VEL
LIN {X 0,Y 496.027,Z 977.884,A -85,B 0,C 180,E1 22728.578,E2 22728.578} C_VEL
LIN {X 0,Y 496.188,Z 971.432,A -85,B 0,C 180,E1 22725.954,E2 22725.954} C_VEL
LIN {X 0,Y 496.499,Z 963.338,A -85,B 0,C 180,E1 22723.363,E2 22723.363} C_VEL
LIN {X 0,Y 497.004,Z 953.528,A -85,B 0,C 180,E1 22720.773,E2 22720.773} C_VEL
LIN {X 0,Y 497.74,Z 941.972,A -85,B 0,C 180,E1 22718.222,E2 22718.222} C_VEL
LIN {X 0,Y 498.754,Z 928.502,A -85,B 0,C 180,E1 22715.688,E2 22715.688} C_VEL
LIN {X 0,Y 500.012,Z 913.65,A -85,B 0,C 180,E1 22713.292,E2 22713.292} C_VEL
LIN {X 0,Y 501.462,Z 897.856,A -85,B 0,C 180,E1 22711.093,E2 22711.093} C_VEL
LIN {X 0,Y 503.171,Z 880.595,A -85,B 0,C 180,E1 22709.003,E2 22709.003} C_VEL
LIN {X 0,Y 504.968,Z 862.37,A -85,B 0,C 180,E1 22707.092,E2 22707.092} C_VEL
LIN {X 0,Y 506.909,Z 843.006,A -85,B 0,C 180,E1 22705.343,E2 22705.343} C_VEL
LIN {X 0,Y 508.913,Z 821.908,A -85,B 0,C 180,E1 22703.714,E2 22703.714} C_VEL
LIN {X 0,Y 510.872,Z 800.318,A -85,B 0,C 180,E1 22702.315,E2 22702.315} C_VEL
LIN {X 0,Y 512.562,Z 779.293,A -85,B 0,C 180,E1 22701.179,E2 22701.179} C_VEL
LIN {X 0,Y 514.139,Z 756.845,A -85,B 0,C 180,E1 22700.197,E2 22700.197} C_VEL
LIN {X 0,Y 515.496,Z 734.117,A -85,B 0,C 180,E1 22699.427,E2 22699.427} C_VEL
LIN {X 0,Y 516.464,Z 711.298,A -85,B 0,C 180,E1 22698.867,E2 22698.867} C_VEL
LIN {X 0,Y 517.857,Z 636.472,A -85,B 0,C 180,E1 22697.635,E2 22697.635} C_VEL
LIN {X 0,Y 521.683,Z 429.085,A -85,B 0,C 180,E1 22694.226,E2 22694.226} C_VEL
LIN {X 0,Y 522.065,Z 405.997,A -85,B 0,C 180,E1 22693.827,E2 22693.827} C_VEL
LIN {X 0,Y 510.537,Z 389.307,A -85,B 0,C 180,E1 22692.211,E2 22692.211} C_VEL
LIN {X 0,Y 503.519,Z 379.594,A -85,B 0,C 180,E1 22691.158,E2 22691.158} C_VEL
LIN {X 0,Y 500.768,Z 375.625,A -85,B 0,C 180,E1 22690.728,E2 22690.728} C_VEL
LIN {X 0,Y 499.763,Z 374.461,A -85,B 0,C 180,E1 22690.575,E2 22690.575} C_VEL
LIN {X 0,Y 497.473,Z 371.587,A -85,B 0,C 180,E1 22690.217,E2 22690.217} C_VEL
LIN {X 0,Y 496.867,Z 369.789,A -85,B 0,C 180,E1 22690.027,E2 22690.027} C_VEL
LIN {X 0,Y 496.763,Z 369.181,A -85,B 0,C 180,E1 22689.734,E2 22689.734} C_VEL
LIN {X 0,Y 496.767,Z 369.166,A -85,B 0,C 180,E1 22686.117,E2 22686.117} C_VEL
LIN {X 0,Y 496.76,Z 369.167,A -85,B 0,C 180,E1 22682.538,E2 22682.538} C_VEL
LIN {X 0,Y 496.769,Z 369.167,A -85,B 0,C 180,E1 22678.962,E2 22678.962} C_VEL
LIN {X 0,Y 496.745,Z 369.163,A -85,B 0,C 180,E1 22675.382,E2 22675.382} C_VEL
LIN {X 0,Y 496.752,Z 369.169,A -85,B 0,C 180,E1 22671.784,E2 22671.784} C_VEL
LIN {X 0,Y 496.77,Z 369.17,A -85,B 0,C 180,E1 22668.271,E2 22668.271} C_VEL
LIN {X 0,Y 496.741,Z 369.168,A -85,B 0,C 180,E1 22664.831,E2 22664.831} C_VEL
LIN {X 0,Y 496.728,Z 369.172,A -85,B 0,C 180,E1 22661.335,E2 22661.335} C_VEL
LIN {X 0,Y 496.771,Z 369.17,A -85,B 0,C 180,E1 22657.891,E2 22657.891} C_VEL
LIN {X 0,Y 496.741,Z 369.172,A -85,B 0,C 180,E1 22654.392,E2 22654.392} C_VEL
LIN {X 0,Y 496.707,Z 369.17,A -85,B 0,C 180,E1 22650.98,E2 22650.98} C_VEL
LIN {X 0,Y 496.749,Z 369.166,A -85,B 0,C 180,E1 22647.629,E2 22647.629} C_VEL
LIN {X 0,Y 496.718,Z 369.177,A -85,B 0,C 180,E1 22644.217,E2 22644.217} C_VEL
LIN {X 0,Y 496.689,Z 369.174,A -85,B 0,C 180,E1 22640.796,E2 22640.796} C_VEL
LIN {X 0,Y 496.783,Z 369.452,A -85,B 0,C 180,E1 22639.795,E2 22639.795} C_VEL
LIN {X 0,Y 498.411,Z 373.208,A -85,B 0,C 180,E1 22639.158,E2 22639.158} C_VEL
LIN {X 0,Y 503.53,Z 383.615,A -85,B 0,C 180,E1 22637.536,E2 22637.536} C_VEL
LIN {X 0,Y 506.249,Z 389.014,A -85,B 0,C 180,E1 22636.78,E2 22636.78} C_VEL
LIN {X 0,Y 521.671,Z 412.741,A -85,B 0,C 180,E1 22634.561,E2 22634.561} C_VEL
LIN {X 0,Y 522.311,Z 417.309,A -85,B 0,C 180,E1 22634.405,E2 22634.405} C_VEL
LIN {X 0,Y 518.494,Z 625.577,A -85,B 0,C 180,E1 22630.973,E2 22630.973} C_VEL
LIN {X 0,Y 516.497,Z 739.86,A -85,B 0,C 180,E1 22629.115,E2 22629.115} C_VEL
LIN {X 0,Y 515.514,Z 762.897,A -85,B 0,C 180,E1 22628.557,E2 22628.557} C_VEL
LIN {X 0,Y 514.414,Z 782.568,A -85,B 0,C 180,E1 22627.914,E2 22627.914} C_VEL
LIN {X 0,Y 512.843,Z 805.185,A -85,B 0,C 180,E1 22626.97,E2 22626.97} C_VEL
LIN {X 0,Y 511.268,Z 825.419,A -85,B 0,C 180,E1 22625.925,E2 22625.925} C_VEL
LIN {X 0,Y 509.447,Z 846.301,A -85,B 0,C 180,E1 22624.626,E2 22624.626} C_VEL
LIN {X 0,Y 507.603,Z 865.79,A -85,B 0,C 180,E1 22623.204,E2 22623.204} C_VEL
LIN {X 0,Y 505.71,Z 885.015,A -85,B 0,C 180,E1 22621.555,E2 22621.555} C_VEL
LIN {X 0,Y 503.887,Z 903.427,A -85,B 0,C 180,E1 22619.743,E2 22619.743} C_VEL
LIN {X 0,Y 502.17,Z 920.599,A -85,B 0,C 180,E1 22617.772,E2 22617.772} C_VEL
LIN {X 0,Y 500.565,Z 937.432,A -85,B 0,C 180,E1 22615.562,E2 22615.562} C_VEL
LIN {X 0,Y 499.285,Z 951.956,A -85,B 0,C 180,E1 22613.363,E2 22613.363} C_VEL
LIN {X 0,Y 498.175,Z 965.804,A -85,B 0,C 180,E1 22610.934,E2 22610.934} C_VEL
LIN {X 0,Y 497.354,Z 977.712,A -85,B 0,C 180,E1 22608.523,E2 22608.523} C_VEL
LIN {X 0,Y 496.736,Z 988.141,A -85,B 0,C 180,E1 22606.01,E2 22606.01} C_VEL
LIN {X 0,Y 496.328,Z 997.271,A -85,B 0,C 180,E1 22603.398,E2 22603.398} C_VEL
LIN {X 0,Y 496.093,Z 1003.976,A -85,B 0,C 180,E1 22601.031,E2 22601.031} C_VEL
LIN {X 0,Y 495.983,Z 1010.01,A -85,B 0,C 180,E1 22598.348,E2 22598.348} C_VEL
LIN {X 0,Y 495.915,Z 1013.955,A -85,B 0,C 180,E1 22595.905,E2 22595.905} C_VEL
LIN {X 0,Y 495.886,Z 1016.713,A -85,B 0,C 180,E1 22593.355,E2 22593.355} C_VEL
LIN {X 0,Y 495.89,Z 1017.827,A -85,B 0,C 180,E1 22590.927,E2 22590.927} C_VEL
LIN {X 0,Y 495.909,Z 1017.714,A -85,B 0,C 180,E1 22588.501,E2 22588.501} C_VEL
LIN {X 0,Y 495.913,Z 1015.959,A -85,B 0,C 180,E1 22585.841,E2 22585.841} C_VEL
LIN {X 0,Y 495.935,Z 1013.005,A -85,B 0,C 180,E1 22583.404,E2 22583.404} C_VEL
LIN {X 0,Y 496.009,Z 1008.09,A -85,B 0,C 180,E1 22580.723,E2 22580.723} C_VEL
LIN {X 0,Y 496.16,Z 1002.139,A -85,B 0,C 180,E1 22578.26,E2 22578.26} C_VEL
LIN {X 0,Y 496.457,Z 994.066,A -85,B 0,C 180,E1 22575.632,E2 22575.632} C_VEL
LIN {X 0,Y 496.917,Z 984.933,A -85,B 0,C 180,E1 22573.161,E2 22573.161} C_VEL
LIN {X 0,Y 497.601,Z 973.745,A -85,B 0,C 180,E1 22570.641,E2 22570.641} C_VEL
LIN {X 0,Y 498.521,Z 961.25,A -85,B 0,C 180,E1 22568.219,E2 22568.219} C_VEL
LIN {X 0,Y 499.672,Z 947.373,A -85,B 0,C 180,E1 22565.912,E2 22565.912} C_VEL
LIN {X 0,Y 501.148,Z 931.218,A -85,B 0,C 180,E1 22563.586,E2 22563.586} C_VEL
LIN {X 0,Y 502.778,Z 914.567,A -85,B 0,C 180,E1 22561.497,E2 22561.497} C_VEL
LIN {X 0,Y 504.464,Z 897.433,A -85,B 0,C 180,E1 22559.646,E2 22559.646} C_VEL
LIN {X 0,Y 506.363,Z 878.501,A -85,B 0,C 180,E1 22557.854,E2 22557.854} C_VEL
LIN {X 0,Y 508.197,Z 859.649,A -85,B 0,C 180,E1 22556.328,E2 22556.328} C_VEL
LIN {X 0,Y 510.099,Z 838.909,A -85,B 0,C 180,E1 22554.885,E2 22554.885} C_VEL
LIN {X 0,Y 511.81,Z 818.758,A -85,B 0,C 180,E1 22553.711,E2 22553.711} C_VEL
LIN {X 0,Y 513.515,Z 796.256,A -85,B 0,C 180,E1 22552.632,E2 22552.632} C_VEL
LIN {X 0,Y 514.78,Z 776.354,A -85,B 0,C 180,E1 22551.865,E2 22551.865} C_VEL
LIN {X 0,Y 515.984,Z 752.256,A -85,B 0,C 180,E1 22551.158,E2 22551.158} C_VEL
LIN {X 0,Y 516.795,Z 729.589,A -85,B 0,C 180,E1 22550.697,E2 22550.697} C_VEL
LIN {X 0,Y 520.427,Z 519.935,A -85,B 0,C 180,E1 22547.292,E2 22547.292} C_VEL
LIN {X 0,Y 522.223,Z 415.374,A -85,B 0,C 180,E1 22545.538,E2 22545.538} C_VEL
LIN {X 0,Y 521.405,Z 412.278,A -85,B 0,C 180,E1 22545.391,E2 22545.391} C_VEL
LIN {X 0,Y 506.483,Z 389.432,A -85,B 0,C 180,E1 22543.237,E2 22543.237} C_VEL
LIN {X 0,Y 500.442,Z 377.322,A -85,B 0,C 180,E1 22541.4,E2 22541.4} C_VEL
LIN {X 0,Y 496.917,Z 370.019,A -85,B 0,C 180,E1 22540.232,E2 22540.232} C_VEL
LIN {X 0,Y 496.773,Z 369.348,A -85,B 0,C 180,E1 22540.095,E2 22540.095} C_VEL
LIN {X 0,Y 496.704,Z 369.167,A -85,B 0,C 180,E1 22536.766,E2 22536.766} C_VEL
LIN {X 0,Y 496.693,Z 369.173,A -85,B 0,C 180,E1 22533.336,E2 22533.336} C_VEL
LIN {X 0,Y 496.753,Z 369.138,A -85,B 0,C 180,E1 22529.945,E2 22529.945} C_VEL
LIN {X 0,Y 496.689,Z 369.176,A -85,B 0,C 180,E1 22526.657,E2 22526.657} C_VEL
LIN {X 0,Y 496.693,Z 369.169,A -85,B 0,C 180,E1 22523.093,E2 22523.093} C_VEL
LIN {X 0,Y 496.751,Z 369.167,A -85,B 0,C 180,E1 22519.764,E2 22519.764} C_VEL
LIN {X 0,Y 496.696,Z 369.172,A -85,B 0,C 180,E1 22516.369,E2 22516.369} C_VEL
LIN {X 0,Y 496.704,Z 369.174,A -85,B 0,C 180,E1 22512.793,E2 22512.793} C_VEL
LIN {X 0,Y 496.761,Z 369.171,A -85,B 0,C 180,E1 22509.383,E2 22509.383} C_VEL
LIN {X 0,Y 496.707,Z 369.174,A -85,B 0,C 180,E1 22506.008,E2 22506.008} C_VEL
LIN {X 0,Y 496.708,Z 369.172,A -85,B 0,C 180,E1 22502.422,E2 22502.422} C_VEL
LIN {X 0,Y 496.77,Z 369.168,A -85,B 0,C 180,E1 22499.077,E2 22499.077} C_VEL
LIN {X 0,Y 496.721,Z 369.174,A -85,B 0,C 180,E1 22495.613,E2 22495.613} C_VEL
LIN {X 0,Y 496.716,Z 369.171,A -85,B 0,C 180,E1 22492.132,E2 22492.132} C_VEL
LIN {X 0,Y 496.771,Z 369.168,A -85,B 0,C 180,E1 22488.741,E2 22488.741} C_VEL
LIN {X 0,Y 496.728,Z 369.172,A -85,B 0,C 180,E1 22485.308,E2 22485.308} C_VEL
LIN {X 0,Y 496.724,Z 369.17,A -85,B 0,C 180,E1 22481.806,E2 22481.806} C_VEL
LIN {X 0,Y 496.775,Z 369.168,A -85,B 0,C 180,E1 22478.387,E2 22478.387} C_VEL
LIN {X 0,Y 496.748,Z 369.17,A -85,B 0,C 180,E1 22474.868,E2 22474.868} C_VEL
LIN {X 0,Y 496.727,Z 369.17,A -85,B 0,C 180,E1 22471.347,E2 22471.347} C_VEL
LIN {X 0,Y 496.765,Z 369.167,A -85,B 0,C 180,E1 22467.902,E2 22467.902} C_VEL
LIN {X 0,Y 496.764,Z 369.171,A -85,B 0,C 180,E1 22464.397,E2 22464.397} C_VEL
LIN {X 0,Y 496.733,Z 369.17,A -85,B 0,C 180,E1 22460.947,E2 22460.947} C_VEL
LIN {X 0,Y 496.758,Z 369.166,A -85,B 0,C 180,E1 22457.442,E2 22457.442} C_VEL
LIN {X 0,Y 496.769,Z 369.164,A -85,B 0,C 180,E1 22453.899,E2 22453.899} C_VEL
LIN {X 0,Y 496.747,Z 369.168,A -85,B 0,C 180,E1 22450.395,E2 22450.395} C_VEL
LIN {X 0,Y 496.744,Z 369.164,A -85,B 0,C 180,E1 22446.764,E2 22446.764} C_VEL
LIN {X 0,Y 496.757,Z 369.169,A -85,B 0,C 180,E1 22446.087,E2 22446.087} C_VEL
LIN {X 0,Y 495.788,Z 369.302,A -85,B 0,C 180,E1 22445.199,E2 22445.199} C_VEL
LIN {X 0,Y 489.333,Z 370.097,A -85,B 0,C 180,E1 22442.701,E2 22442.701} C_VEL
LIN {X 0,Y 488.817,Z 370.149,A -85,B 0,C 180,E1 22442.049,E2 22442.049} C_VEL
LIN {X 0,Y 488.812,Z 370.157,A -85,B 0,C 180,E1 22438.41,E2 22438.41} C_VEL
LIN {X 0,Y 488.824,Z 370.138,A -85,B 0,C 180,E1 22434.787,E2 22434.787} C_VEL
LIN {X 0,Y 488.819,Z 370.132,A -85,B 0,C 180,E1 22431.222,E2 22431.222} C_VEL
LIN {X 0,Y 488.817,Z 370.133,A -85,B 0,C 180,E1 22427.741,E2 22427.741} C_VEL
LIN {X 0,Y 488.852,Z 370.357,A -85,B 0,C 180,E1 22426.941,E2 22426.941} C_VEL
LIN {X 0,Y 489.247,Z 371.884,A -85,B 0,C 180,E1 22426.702,E2 22426.702} C_VEL
LIN {X 0,Y 491.127,Z 374.831,A -85,B 0,C 180,E1 22426.383,E2 22426.383} C_VEL
LIN {X 0,Y 492.785,Z 376.491,A -85,B 0,C 180,E1 22426.13,E2 22426.13} C_VEL
LIN {X 0,Y 495.43,Z 380.428,A -85,B 0,C 180,E1 22425.705,E2 22425.705} C_VEL
LIN {X 0,Y 497.134,Z 382.616,A -85,B 0,C 180,E1 22425.443,E2 22425.443} C_VEL
LIN {X 0,Y 507.803,Z 397.385,A -85,B 0,C 180,E1 22423.841,E2 22423.841} C_VEL
LIN {X 0,Y 516.316,Z 410.028,A -85,B 0,C 180,E1 22422.623,E2 22422.623} C_VEL
LIN {X 0,Y 511.911,Z 627.706,A -85,B 0,C 180,E1 22418.997,E2 22418.997} C_VEL
LIN {X 0,Y 510.219,Z 711.633,A -85,B 0,C 180,E1 22417.602,E2 22417.602} C_VEL
LIN {X 0,Y 509.182,Z 734.438,A -85,B 0,C 180,E1 22417.036,E2 22417.036} C_VEL
LIN {X 0,Y 507.758,Z 757.024,A -85,B 0,C 180,E1 22416.264,E2 22416.264} C_VEL
LIN {X 0,Y 506.057,Z 779.483,A -85,B 0,C 180,E1 22415.274,E2 22415.274} C_VEL
LIN {X 0,Y 504.247,Z 800.264,A -85,B 0,C 180,E1 22414.14,E2 22414.14} C_VEL
LIN {X 0,Y 502.158,Z 821.737,A -85,B 0,C 180,E1 22412.736,E2 22412.736} C_VEL
LIN {X 0,Y 500.03,Z 842.32,A -85,B 0,C 180,E1 22411.136,E2 22411.136} C_VEL
LIN {X 0,Y 497.862,Z 862.374,A -85,B 0,C 180,E1 22409.307,E2 22409.307} C_VEL
LIN {X 0,Y 495.81,Z 881.378,A -85,B 0,C 180,E1 22407.281,E2 22407.281} C_VEL
LIN {X 0,Y 493.925,Z 898.856,A -85,B 0,C 180,E1 22405.12,E2 22405.12} C_VEL
LIN {X 0,Y 492.352,Z 914.55,A -85,B 0,C 180,E1 22402.881,E2 22402.881} C_VEL
LIN {X 0,Y 491.016,Z 928.994,A -85,B 0,C 180,E1 22400.503,E2 22400.503} C_VEL
LIN {X 0,Y 489.921,Z 942.128,A -85,B 0,C 180,E1 22397.982,E2 22397.982} C_VEL
LIN {X 0,Y 489.122,Z 953.479,A -85,B 0,C 180,E1 22395.435,E2 22395.435} C_VEL
LIN {X 0,Y 488.572,Z 963.108,A -85,B 0,C 180,E1 22392.858,E2 22392.858} C_VEL
LIN {X 0,Y 488.217,Z 971.167,A -85,B 0,C 180,E1 22390.247,E2 22390.247} C_VEL
LIN {X 0,Y 488.032,Z 977.645,A -85,B 0,C 180,E1 22387.598,E2 22387.598} C_VEL
LIN {X 0,Y 487.943,Z 982.654,A -85,B 0,C 180,E1 22384.899,E2 22384.899} C_VEL
LIN {X 0,Y 487.893,Z 985.913,A -85,B 0,C 180,E1 22382.274,E2 22382.274} C_VEL
LIN {X 0,Y 487.886,Z 987.635,A -85,B 0,C 180,E1 22379.723,E2 22379.723} C_VEL
LIN {X 0,Y 487.901,Z 987.866,A -85,B 0,C 180,E1 22377.105,E2 22377.105} C_VEL
LIN {X 0,Y 487.912,Z 986.583,A -85,B 0,C 180,E1 22374.407,E2 22374.407} C_VEL
LIN {X 0,Y 487.92,Z 983.668,A -85,B 0,C 180,E1 22371.708,E2 22371.708} C_VEL
LIN {X 0,Y 487.99,Z 979.181,A -85,B 0,C 180,E1 22369.028,E2 22369.028} C_VEL
LIN {X 0,Y 488.148,Z 973.336,A -85,B 0,C 180,E1 22366.477,E2 22366.477} C_VEL
LIN {X 0,Y 488.48,Z 965.377,A -85,B 0,C 180,E1 22363.732,E2 22363.732} C_VEL
LIN {X 0,Y 488.975,Z 956.007,A -85,B 0,C 180,E1 22361.118,E2 22361.118} C_VEL
LIN {X 0,Y 489.769,Z 944.238,A -85,B 0,C 180,E1 22358.376,E2 22358.376} C_VEL
LIN {X 0,Y 490.836,Z 931.03,A -85,B 0,C 180,E1 22355.777,E2 22355.777} C_VEL
LIN {X 0,Y 492.131,Z 916.798,A -85,B 0,C 180,E1 22353.379,E2 22353.379} C_VEL
LIN {X 0,Y 493.807,Z 900.054,A -85,B 0,C 180,E1 22350.951,E2 22350.951} C_VEL
LIN {X 0,Y 495.712,Z 882.298,A -85,B 0,C 180,E1 22348.735,E2 22348.735} C_VEL
LIN {X 0,Y 497.702,Z 863.805,A -85,B 0,C 180,E1 22346.744,E2 22346.744} C_VEL
LIN {X 0,Y 499.876,Z 843.821,A -85,B 0,C 180,E1 22344.901,E2 22344.901} C_VEL
LIN {X 0,Y 501.992,Z 823.36,A -85,B 0,C 180,E1 22343.289,E2 22343.289} C_VEL
LIN {X 0,Y 504.063,Z 802.384,A -85,B 0,C 180,E1 22341.896,E2 22341.896} C_VEL
LIN {X 0,Y 505.934,Z 781.146,A -85,B 0,C 180,E1 22340.717,E2 22340.717} C_VEL
LIN {X 0,Y 507.659,Z 758.344,A -85,B 0,C 180,E1 22339.697,E2 22339.697} C_VEL
LIN {X 0,Y 509.131,Z 735.262,A -85,B 0,C 180,E1 22338.9,E2 22338.9} C_VEL
LIN {X 0,Y 510.171,Z 712.795,A -85,B 0,C 180,E1 22338.334,E2 22338.334} C_VEL
LIN {X 0,Y 511.373,Z 655.826,A -85,B 0,C 180,E1 22337.375,E2 22337.375} C_VEL
LIN {X 0,Y 515.492,Z 448.711,A -85,B 0,C 180,E1 22333.94,E2 22333.94} C_VEL
LIN {X 0,Y 516.207,Z 409.476,A -85,B 0,C 180,E1 22333.255,E2 22333.255} C_VEL
LIN {X 0,Y 503.295,Z 390.931,A -85,B 0,C 180,E1 22331.372,E2 22331.372} C_VEL
LIN {X 0,Y 498.585,Z 384.677,A -85,B 0,C 180,E1 22330.647,E2 22330.647} C_VEL
LIN {X 0,Y 495.921,Z 380.878,A -85,B 0,C 180,E1 22330.22,E2 22330.22} C_VEL
LIN {X 0,Y 493.161,Z 377.143,A -85,B 0,C 180,E1 22329.774,E2 22329.774} C_VEL
LIN {X 0,Y 492.23,Z 375.753,A -85,B 0,C 180,E1 22329.618,E2 22329.618} C_VEL
LIN {X 0,Y 489.761,Z 373.035,A -85,B 0,C 180,E1 22329.222,E2 22329.222} C_VEL
LIN {X 0,Y 488.896,Z 370.662,A -85,B 0,C 180,E1 22328.942,E2 22328.942} C_VEL
LIN {X 0,Y 488.817,Z 370.157,A -85,B 0,C 180,E1 22328.588,E2 22328.588} C_VEL
LIN {X 0,Y 488.825,Z 370.159,A -85,B 0,C 180,E1 22325.034,E2 22325.034} C_VEL
LIN {X 0,Y 488.814,Z 370.159,A -85,B 0,C 180,E1 22321.524,E2 22321.524} C_VEL
LIN {X 0,Y 488.823,Z 370.154,A -85,B 0,C 180,E1 22318.008,E2 22318.008} C_VEL
LIN {X 0,Y 488.829,Z 370.153,A -85,B 0,C 180,E1 22314.366,E2 22314.366} C_VEL
LIN {X 0,Y 488.821,Z 370.158,A -85,B 0,C 180,E1 22310.82,E2 22310.82} C_VEL
LIN {X 0,Y 488.795,Z 370.161,A -85,B 0,C 180,E1 22307.237,E2 22307.237} C_VEL
LIN {X 0,Y 488.811,Z 370.16,A -85,B 0,C 180,E1 22303.726,E2 22303.726} C_VEL
LIN {X 0,Y 488.832,Z 370.158,A -85,B 0,C 180,E1 22300.152,E2 22300.152} C_VEL
LIN {X 0,Y 488.788,Z 370.161,A -85,B 0,C 180,E1 22296.706,E2 22296.706} C_VEL
LIN {X 0,Y 488.777,Z 370.163,A -85,B 0,C 180,E1 22293.115,E2 22293.115} C_VEL
LIN {X 0,Y 488.812,Z 370.158,A -85,B 0,C 180,E1 22289.654,E2 22289.654} C_VEL
LIN {X 0,Y 488.793,Z 370.16,A -85,B 0,C 180,E1 22286.153,E2 22286.153} C_VEL
LIN {X 0,Y 488.753,Z 370.163,A -85,B 0,C 180,E1 22282.732,E2 22282.732} C_VEL
LIN {X 0,Y 488.788,Z 370.425,A -85,B 0,C 180,E1 22280.796,E2 22280.796} C_VEL
LIN {X 0,Y 490.24,Z 373.893,A -85,B 0,C 180,E1 22280.178,E2 22280.178} C_VEL
LIN {X 0,Y 491.356,Z 375.83,A -85,B 0,C 180,E1 22279.83,E2 22279.83} C_VEL
LIN {X 0,Y 497.551,Z 388.11,A -85,B 0,C 180,E1 22277.88,E2 22277.88} C_VEL
LIN {X 0,Y 511.486,Z 409.473,A -85,B 0,C 180,E1 22275.744,E2 22275.744} C_VEL
LIN {X 0,Y 516.499,Z 417.751,A -85,B 0,C 180,E1 22275.023,E2 22275.023} C_VEL
LIN {X 0,Y 512.707,Z 606.696,A -85,B 0,C 180,E1 22271.857,E2 22271.857} C_VEL
LIN {X 0,Y 510.18,Z 740.289,A -85,B 0,C 180,E1 22269.662,E2 22269.662} C_VEL
LIN {X 0,Y 509.143,Z 763.233,A -85,B 0,C 180,E1 22269.1,E2 22269.1} C_VEL
LIN {X 0,Y 507.966,Z 783.602,A -85,B 0,C 180,E1 22268.432,E2 22268.432} C_VEL
LIN {X 0,Y 506.392,Z 805.054,A -85,B 0,C 180,E1 22267.528,E2 22267.528} C_VEL
LIN {X 0,Y 504.636,Z 825.841,A -85,B 0,C 180,E1 22266.446,E2 22266.446} C_VEL
LIN {X 0,Y 502.617,Z 847.197,A -85,B 0,C 180,E1 22265.095,E2 22265.095} C_VEL
LIN {X 0,Y 500.645,Z 866.597,A -85,B 0,C 180,E1 22263.658,E2 22263.658} C_VEL
LIN {X 0,Y 498.563,Z 885.904,A -85,B 0,C 180,E1 22261.97,E2 22261.97} C_VEL
LIN {X 0,Y 496.552,Z 904.545,A -85,B 0,C 180,E1 22260.094,E2 22260.094} C_VEL
LIN {X 0,Y 494.752,Z 921.105,A -85,B 0,C 180,E1 22258.159,E2 22258.159} C_VEL
LIN {X 0,Y 492.962,Z 938.279,A -85,B 0,C 180,E1 22255.856,E2 22255.856} C_VEL
LIN {X 0,Y 491.518,Z 953.492,A -85,B 0,C 180,E1 22253.5,E2 22253.5} C_VEL
LIN {X 0,Y 490.321,Z 967.072,A -85,B 0,C 180,E1 22251.035,E2 22251.035} C_VEL
LIN {X 0,Y 489.405,Z 979.278,A -85,B 0,C 180,E1 22248.464,E2 22248.464} C_VEL
LIN {X 0,Y 488.784,Z 989.057,A -85,B 0,C 180,E1 22246.034,E2 22246.034} C_VEL
LIN {X 0,Y 488.337,Z 998.341,A -85,B 0,C 180,E1 22243.26,E2 22243.26} C_VEL
LIN {X 0,Y 488.099,Z 1004.859,A -85,B 0,C 180,E1 22240.866,E2 22240.866} C_VEL
LIN {X 0,Y 487.98,Z 1010.63,A -85,B 0,C 180,E1 22238.13,E2 22238.13} C_VEL
LIN {X 0,Y 487.912,Z 1014.433,A -85,B 0,C 180,E1 22235.648,E2 22235.648} C_VEL
LIN {X 0,Y 487.89,Z 1016.984,A -85,B 0,C 180,E1 22232.94,E2 22232.94} C_VEL
LIN {X 0,Y 487.885,Z 1017.894,A -85,B 0,C 180,E1 22230.59,E2 22230.59} C_VEL
LIN {X 0,Y 487.913,Z 1017.394,A -85,B 0,C 180,E1 22227.772,E2 22227.772} C_VEL
LIN {X 0,Y 487.906,Z 1015.504,A -85,B 0,C 180,E1 22225.301,E2 22225.301} C_VEL
LIN {X 0,Y 487.931,Z 1011.88,A -85,B 0,C 180,E1 22222.586,E2 22222.586} C_VEL
LIN {X 0,Y 488.017,Z 1007.346,A -85,B 0,C 180,E1 22220.222,E2 22220.222} C_VEL
LIN {X 0,Y 488.242,Z 1000.83,A -85,B 0,C 180,E1 22217.587,E2 22217.587} C_VEL
LIN {X 0,Y 488.592,Z 992.95,A -85,B 0,C 180,E1 22215.061,E2 22215.061} C_VEL
LIN {X 0,Y 489.198,Z 982.339,A -85,B 0,C 180,E1 22212.258,E2 22212.258} C_VEL
LIN {X 0,Y 489.978,Z 971.435,A -85,B 0,C 180,E1 22209.83,E2 22209.83} C_VEL
LIN {X 0,Y 491.056,Z 958.475,A -85,B 0,C 180,E1 22207.371,E2 22207.371} C_VEL
LIN {X 0,Y 492.405,Z 944.239,A -85,B 0,C 180,E1 22205.021,E2 22205.021} C_VEL
LIN {X 0,Y 493.961,Z 928.439,A -85,B 0,C 180,E1 22202.781,E2 22202.781} C_VEL
LIN {X 0,Y 495.924,Z 910.152,A -85,B 0,C 180,E1 22200.536,E2 22200.536} C_VEL
LIN {X 0,Y 497.86,Z 892.564,A -85,B 0,C 180,E1 22198.662,E2 22198.662} C_VEL
LIN {X 0,Y 499.912,Z 873.365,A -85,B 0,C 180,E1 22196.911,E2 22196.911} C_VEL
LIN {X 0,Y 501.985,Z 853.574,A -85,B 0,C 180,E1 22195.347,E2 22195.347} C_VEL
LIN {X 0,Y 503.897,Z 833.882,A -85,B 0,C 180,E1 22194.037,E2 22194.037} C_VEL
LIN {X 0,Y 505.799,Z 812.767,A -85,B 0,C 180,E1 22192.848,E2 22192.848} C_VEL
LIN {X 0,Y 507.326,Z 792.528,A -85,B 0,C 180,E1 22191.917,E2 22191.917} C_VEL
LIN {X 0,Y 508.836,Z 769.346,A -85,B 0,C 180,E1 22191.077,E2 22191.077} C_VEL
LIN {X 0,Y 509.858,Z 748.784,A -85,B 0,C 180,E1 22190.521,E2 22190.521} C_VEL
LIN {X 0,Y 510.697,Z 721.521,A -85,B 0,C 180,E1 22190.004,E2 22190.004} C_VEL
LIN {X 0,Y 514.58,Z 516.749,A -85,B 0,C 180,E1 22186.637,E2 22186.637} C_VEL
LIN {X 0,Y 516.468,Z 417.304,A -85,B 0,C 180,E1 22184.95,E2 22184.95} C_VEL
LIN {X 0,Y 501.537,Z 394.363,A -85,B 0,C 180,E1 22182.751,E2 22182.751} C_VEL
LIN {X 0,Y 497.783,Z 388.69,A -85,B 0,C 180,E1 22182.134,E2 22182.134} C_VEL
LIN {X 0,Y 492.21,Z 377.728,A -85,B 0,C 180,E1 22180.387,E2 22180.387} C_VEL
LIN {X 0,Y 490.463,Z 374.14,A -85,B 0,C 180,E1 22179.8,E2 22179.8} C_VEL
LIN {X 0,Y 488.807,Z 370.508,A -85,B 0,C 180,E1 22179.18,E2 22179.18} C_VEL
LIN {X 0,Y 488.816,Z 370.14,A -85,B 0,C 180,E1 22178.15,E2 22178.15} C_VEL
LIN {X 0,Y 488.764,Z 370.131,A -85,B 0,C 180,E1 22174.659,E2 22174.659} C_VEL
LIN {X 0,Y 488.748,Z 370.141,A -85,B 0,C 180,E1 22171.169,E2 22171.169} C_VEL
LIN {X 0,Y 488.804,Z 370.16,A -85,B 0,C 180,E1 22167.799,E2 22167.799} C_VEL
LIN {X 0,Y 488.761,Z 370.166,A -85,B 0,C 180,E1 22164.408,E2 22164.408} C_VEL
LIN {X 0,Y 488.751,Z 370.163,A -85,B 0,C 180,E1 22160.852,E2 22160.852} C_VEL
LIN {X 0,Y 488.797,Z 370.156,A -85,B 0,C 180,E1 22157.376,E2 22157.376} C_VEL
LIN {X 0,Y 488.772,Z 370.157,A -85,B 0,C 180,E1 22154.089,E2 22154.089} C_VEL
LIN {X 0,Y 488.761,Z 370.16,A -85,B 0,C 180,E1 22150.609,E2 22150.609} C_VEL
LIN {X 0,Y 488.815,Z 370.157,A -85,B 0,C 180,E1 22147.167,E2 22147.167} C_VEL
LIN {X 0,Y 488.782,Z 370.157,A -85,B 0,C 180,E1 22143.753,E2 22143.753} C_VEL
LIN {X 0,Y 488.769,Z 370.16,A -85,B 0,C 180,E1 22140.234,E2 22140.234} C_VEL
LIN {X 0,Y 488.813,Z 370.159,A -85,B 0,C 180,E1 22136.805,E2 22136.805} C_VEL
LIN {X 0,Y 488.802,Z 370.155,A -85,B 0,C 180,E1 22133.304,E2 22133.304} C_VEL
LIN {X 0,Y 488.775,Z 370.157,A -85,B 0,C 180,E1 22129.867,E2 22129.867} C_VEL
LIN {X 0,Y 488.812,Z 370.157,A -85,B 0,C 180,E1 22126.394,E2 22126.394} C_VEL
LIN {X 0,Y 488.821,Z 370.153,A -85,B 0,C 180,E1 22122.869,E2 22122.869} C_VEL
LIN {X 0,Y 488.784,Z 370.153,A -85,B 0,C 180,E1 22119.4,E2 22119.4} C_VEL
LIN {X 0,Y 488.795,Z 370.155,A -85,B 0,C 180,E1 22115.816,E2 22115.816} C_VEL
LIN {X 0,Y 488.836,Z 370.153,A -85,B 0,C 180,E1 22112.321,E2 22112.321} C_VEL
LIN {X 0,Y 488.808,Z 370.153,A -85,B 0,C 180,E1 22108.753,E2 22108.753} C_VEL
LIN {X 0,Y 488.792,Z 370.155,A -85,B 0,C 180,E1 22105.2,E2 22105.2} C_VEL
LIN {X 0,Y 488.827,Z 370.156,A -85,B 0,C 180,E1 22101.701,E2 22101.701} C_VEL
LIN {X 0,Y 488.831,Z 370.158,A -85,B 0,C 180,E1 22098.112,E2 22098.112} C_VEL
LIN {X 0,Y 488.804,Z 370.16,A -85,B 0,C 180,E1 22094.55,E2 22094.55} C_VEL
LIN {X 0,Y 488.804,Z 370.158,A -85,B 0,C 180,E1 22090.881,E2 22090.881} C_VEL
LIN {X 0,Y 488.828,Z 370.15,A -85,B 0,C 180,E1 22087.403,E2 22087.403} C_VEL
LIN {X 0,Y 488.832,Z 370.155,A -85,B 0,C 180,E1 22083.799,E2 22083.799} C_VEL
LIN {X 0,Y 488.817,Z 370.149,A -85,B 0,C 180,E1 22082.049,E2 22082.049} C_VEL
LIN {X 0,Y 487.845,Z 370.257,A -85,B 0,C 180,E1 22081.146,E2 22081.146} C_VEL
LIN {X 0,Y 481.389,Z 371.081,A -85,B 0,C 180,E1 22078.607,E2 22078.607} C_VEL
LIN {X 0,Y 480.883,Z 371.15,A -85,B 0,C 180,E1 22077.945,E2 22077.945} C_VEL
LIN {X 0,Y 480.872,Z 371.135,A -85,B 0,C 180,E1 22074.307,E2 22074.307} C_VEL
LIN {X 0,Y 480.887,Z 371.121,A -85,B 0,C 180,E1 22070.695,E2 22070.695} C_VEL
LIN {X 0,Y 480.892,Z 371.264,A -85,B 0,C 180,E1 22068.043,E2 22068.043} C_VEL
LIN {X 0,Y 481.253,Z 372.742,A -85,B 0,C 180,E1 22067.779,E2 22067.779} C_VEL
LIN {X 0,Y 483.144,Z 375.766,A -85,B 0,C 180,E1 22067.439,E2 22067.439} C_VEL
LIN {X 0,Y 484.907,Z 377.414,A -85,B 0,C 180,E1 22067.159,E2 22067.159} C_VEL
LIN {X 0,Y 487.533,Z 381.402,A -85,B 0,C 180,E1 22066.714,E2 22066.714} C_VEL
LIN {X 0,Y 489.219,Z 383.508,A -85,B 0,C 180,E1 22066.443,E2 22066.443} C_VEL
LIN {X 0,Y 500.502,Z 398.948,A -85,B 0,C 180,E1 22064.682,E2 22064.682} C_VEL
LIN {X 0,Y 510.565,Z 413.556,A -85,B 0,C 180,E1 22063.198,E2 22063.198} C_VEL
LIN {X 0,Y 505.822,Z 629.445,A -85,B 0,C 180,E1 22059.562,E2 22059.562} C_VEL
LIN {X 0,Y 504.013,Z 712.17,A -85,B 0,C 180,E1 22058.169,E2 22058.169} C_VEL
LIN {X 0,Y 502.9,Z 734.846,A -85,B 0,C 180,E1 22057.598,E2 22057.598} C_VEL
LIN {X 0,Y 501.427,Z 757.118,A -85,B 0,C 180,E1 22056.832,E2 22056.832} C_VEL
LIN {X 0,Y 499.636,Z 779.183,A -85,B 0,C 180,E1 22055.855,E2 22055.855} C_VEL
LIN {X 0,Y 497.621,Z 800.823,A -85,B 0,C 180,E1 22054.664,E2 22054.664} C_VEL
LIN {X 0,Y 495.46,Z 821.509,A -85,B 0,C 180,E1 22053.294,E2 22053.294} C_VEL
LIN {X 0,Y 493.144,Z 842.139,A -85,B 0,C 180,E1 22051.678,E2 22051.678} C_VEL
LIN {X 0,Y 490.815,Z 862.252,A -85,B 0,C 180,E1 22049.822,E2 22049.822} C_VEL
LIN {X 0,Y 488.569,Z 881.298,A -85,B 0,C 180,E1 22047.769,E2 22047.769} C_VEL
LIN {X 0,Y 486.58,Z 898.353,A -85,B 0,C 180,E1 22045.637,E2 22045.637} C_VEL
LIN {X 0,Y 484.854,Z 914.11,A -85,B 0,C 180,E1 22043.366,E2 22043.366} C_VEL
LIN {X 0,Y 483.372,Z 928.608,A -85,B 0,C 180,E1 22040.952,E2 22040.952} C_VEL
LIN {X 0,Y 482.159,Z 941.792,A -85,B 0,C 180,E1 22038.393,E2 22038.393} C_VEL
LIN {X 0,Y 481.274,Z 953.158,A -85,B 0,C 180,E1 22035.807,E2 22035.807} C_VEL
LIN {X 0,Y 480.645,Z 963.077,A -85,B 0,C 180,E1 22033.12,E2 22033.12} C_VEL
LIN {X 0,Y 480.258,Z 970.928,A -85,B 0,C 180,E1 22030.54,E2 22030.54} C_VEL
LIN {X 0,Y 480.044,Z 977.457,A -85,B 0,C 180,E1 22027.85,E2 22027.85} C_VEL
LIN {X 0,Y 479.958,Z 982.322,A -85,B 0,C 180,E1 22025.243,E2 22025.243} C_VEL
LIN {X 0,Y 479.891,Z 985.821,A -85,B 0,C 180,E1 22022.446,E2 22022.446} C_VEL
LIN {X 0,Y 479.883,Z 987.589,A -85,B 0,C 180,E1 22019.846,E2 22019.846} C_VEL
LIN {X 0,Y 479.899,Z 987.883,A -85,B 0,C 180,E1 22017.198,E2 22017.198} C_VEL
LIN {X 0,Y 479.912,Z 986.668,A -85,B 0,C 180,E1 22014.457,E2 22014.457} C_VEL
LIN {X 0,Y 479.918,Z 983.881,A -85,B 0,C 180,E1 22011.762,E2 22011.762} C_VEL
LIN {X 0,Y 479.985,Z 979.658,A -85,B 0,C 180,E1 22009.128,E2 22009.128} C_VEL
LIN {X 0,Y 480.165,Z 973.699,A -85,B 0,C 180,E1 22006.427,E2 22006.427} C_VEL
LIN {X 0,Y 480.51,Z 966.01,A -85,B 0,C 180,E1 22003.697,E2 22003.697} C_VEL
LIN {X 0,Y 481.046,Z 956.701,A -85,B 0,C 180,E1 22001.016,E2 22001.016} C_VEL
LIN {X 0,Y 481.917,Z 944.9,A -85,B 0,C 180,E1 21998.191,E2 21998.191} C_VEL
LIN {X 0,Y 483.061,Z 931.882,A -85,B 0,C 180,E1 21995.564,E2 21995.564} C_VEL
LIN {X 0,Y 484.534,Z 917.053,A -85,B 0,C 180,E1 21993.01,E2 21993.01} C_VEL
LIN {X 0,Y 486.307,Z 900.752,A -85,B 0,C 180,E1 21990.6,E2 21990.6} C_VEL
LIN {X 0,Y 488.291,Z 883.763,A -85,B 0,C 180,E1 21988.43,E2 21988.43} C_VEL
LIN {X 0,Y 490.359,Z 866.082,A -85,B 0,C 180,E1 21986.472,E2 21986.472} C_VEL
LIN {X 0,Y 492.678,Z 846.465,A -85,B 0,C 180,E1 21984.604,E2 21984.604} C_VEL
LIN {X 0,Y 494.965,Z 826.108,A -85,B 0,C 180,E1 21982.947,E2 21982.947} C_VEL
LIN {X 0,Y 497.283,Z 804.452,A -85,B 0,C 180,E1 21981.466,E2 21981.466} C_VEL
LIN {X 0,Y 499.39,Z 782.203,A -85,B 0,C 180,E1 21980.205,E2 21980.205} C_VEL
LIN {X 0,Y 501.208,Z 759.935,A -85,B 0,C 180,E1 21979.188,E2 21979.188} C_VEL
LIN {X 0,Y 502.792,Z 736.419,A -85,B 0,C 180,E1 21978.362,E2 21978.362} C_VEL
LIN {X 0,Y 503.909,Z 714.468,A -85,B 0,C 180,E1 21977.793,E2 21977.793} C_VEL
LIN {X 0,Y 504.974,Z 669.808,A -85,B 0,C 180,E1 21977.02,E2 21977.02} C_VEL
LIN {X 0,Y 509.382,Z 464.289,A -85,B 0,C 180,E1 21973.579,E2 21973.579} C_VEL
LIN {X 0,Y 510.481,Z 413.354,A -85,B 0,C 180,E1 21972.691,E2 21972.691} C_VEL
LIN {X 0,Y 498.923,Z 396.64,A -85,B 0,C 180,E1 21970.949,E2 21970.949} C_VEL
LIN {X 0,Y 491.591,Z 386.685,A -85,B 0,C 180,E1 21969.778,E2 21969.778} C_VEL
LIN {X 0,Y 488.073,Z 381.918,A -85,B 0,C 180,E1 21969.195,E2 21969.195} C_VEL
LIN {X 0,Y 485.302,Z 378.081,A -85,B 0,C 180,E1 21968.71,E2 21968.71} C_VEL
LIN {X 0,Y 484.303,Z 376.76,A -85,B 0,C 180,E1 21968.534,E2 21968.534} C_VEL
LIN {X 0,Y 481.865,Z 374.094,A -85,B 0,C 180,E1 21968.112,E2 21968.112} C_VEL
LIN {X 0,Y 481.031,Z 371.974,A -85,B 0,C 180,E1 21967.885,E2 21967.885} C_VEL
LIN {X 0,Y 480.888,Z 371.167,A -85,B 0,C 180,E1 21967.527,E2 21967.527} C_VEL
LIN {X 0,Y 480.879,Z 371.145,A -85,B 0,C 180,E1 21963.815,E2 21963.815} C_VEL
LIN {X 0,Y 480.896,Z 371.141,A -85,B 0,C 180,E1 21960.12,E2 21960.12} C_VEL
LIN {X 0,Y 480.888,Z 371.148,A -85,B 0,C 180,E1 21956.403,E2 21956.403} C_VEL
LIN {X 0,Y 480.894,Z 371.139,A -85,B 0,C 180,E1 21952.714,E2 21952.714} C_VEL
LIN {X 0,Y 480.864,Z 371.147,A -85,B 0,C 180,E1 21949.093,E2 21949.093} C_VEL
LIN {X 0,Y 480.857,Z 371.149,A -85,B 0,C 180,E1 21945.428,E2 21945.428} C_VEL
LIN {X 0,Y 480.882,Z 371.149,A -85,B 0,C 180,E1 21941.828,E2 21941.828} C_VEL
LIN {X 0,Y 480.888,Z 371.148,A -85,B 0,C 180,E1 21938.279,E2 21938.279} C_VEL
LIN {X 0,Y 480.842,Z 371.152,A -85,B 0,C 180,E1 21934.764,E2 21934.764} C_VEL
LIN {X 0,Y 480.832,Z 371.148,A -85,B 0,C 180,E1 21931.1,E2 21931.1} C_VEL
LIN {X 0,Y 480.877,Z 371.141,A -85,B 0,C 180,E1 21927.7,E2 21927.7} C_VEL
LIN {X 0,Y 480.842,Z 371.154,A -85,B 0,C 180,E1 21924.193,E2 21924.193} C_VEL
LIN {X 0,Y 480.91,Z 371.441,A -85,B 0,C 180,E1 21921.833,E2 21921.833} C_VEL
LIN {X 0,Y 482.231,Z 374.762,A -85,B 0,C 180,E1 21921.226,E2 21921.226} C_VEL
LIN {X 0,Y 483.608,Z 377.341,A -85,B 0,C 180,E1 21920.754,E2 21920.754} C_VEL
LIN {X 0,Y 486.064,Z 382.07,A -85,B 0,C 180,E1 21919.921,E2 21919.921} C_VEL
LIN {X 0,Y 489.001,Z 387.729,A -85,B 0,C 180,E1 21919.017,E2 21919.017} C_VEL
LIN {X 0,Y 498.268,Z 401.437,A -85,B 0,C 180,E1 21917.488,E2 21917.488} C_VEL
LIN {X 0,Y 510.776,Z 421.283,A -85,B 0,C 180,E1 21915.588,E2 21915.588} C_VEL
LIN {X 0,Y 506.212,Z 628.93,A -85,B 0,C 180,E1 21912.082,E2 21912.082} C_VEL
LIN {X 0,Y 503.907,Z 740.255,A -85,B 0,C 180,E1 21910.229,E2 21910.229} C_VEL
LIN {X 0,Y 502.794,Z 763.002,A -85,B 0,C 180,E1 21909.666,E2 21909.666} C_VEL
LIN {X 0,Y 501.5,Z 783.891,A -85,B 0,C 180,E1 21908.973,E2 21908.973} C_VEL
LIN {X 0,Y 499.716,Z 806.645,A -85,B 0,C 180,E1 21907.999,E2 21907.999} C_VEL
LIN {X 0,Y 497.82,Z 828.655,A -85,B 0,C 180,E1 21906.838,E2 21906.838} C_VEL
LIN {X 0,Y 495.822,Z 848.094,A -85,B 0,C 180,E1 21905.578,E2 21905.578} C_VEL
LIN {X 0,Y 493.621,Z 868.17,A -85,B 0,C 180,E1 21904.061,E2 21904.061} C_VEL
LIN {X 0,Y 491.394,Z 887.237,A -85,B 0,C 180,E1 21902.355,E2 21902.355} C_VEL
LIN {X 0,Y 489.09,Z 906.763,A -85,B 0,C 180,E1 21900.33,E2 21900.33} C_VEL
LIN {X 0,Y 487.2,Z 923.132,A -85,B 0,C 180,E1 21898.368,E2 21898.368} C_VEL
LIN {X 0,Y 485.372,Z 939.122,A -85,B 0,C 180,E1 21896.16,E2 21896.16} C_VEL
LIN {X 0,Y 483.89,Z 953.492,A -85,B 0,C 180,E1 21893.893,E2 21893.893} C_VEL
LIN {X 0,Y 482.623,Z 966.435,A -85,B 0,C 180,E1 21891.514,E2 21891.514} C_VEL
LIN {X 0,Y 481.597,Z 978.759,A -85,B 0,C 180,E1 21888.9,E2 21888.9} C_VEL
LIN {X 0,Y 480.903,Z 988.597,A -85,B 0,C 180,E1 21886.428,E2 21886.428} C_VEL
LIN {X 0,Y 480.407,Z 997.629,A -85,B 0,C 180,E1 21883.728,E2 21883.728} C_VEL
LIN {X 0,Y 480.131,Z 1004.252,A -85,B 0,C 180,E1 21881.291,E2 21881.291} C_VEL
LIN {X 0,Y 479.994,Z 1010.217,A -85,B 0,C 180,E1 21878.508,E2 21878.508} C_VEL
LIN {X 0,Y 479.921,Z 1014.115,A -85,B 0,C 180,E1 21875.982,E2 21875.982} C_VEL
LIN {X 0,Y 479.885,Z 1016.848,A -85,B 0,C 180,E1 21873.228,E2 21873.228} C_VEL
LIN {X 0,Y 479.887,Z 1017.849,A -85,B 0,C 180,E1 21870.839,E2 21870.839} C_VEL
LIN {X 0,Y 479.907,Z 1017.659,A -85,B 0,C 180,E1 21868.212,E2 21868.212} C_VEL
LIN {X 0,Y 479.908,Z 1015.845,A -85,B 0,C 180,E1 21865.582,E2 21865.582} C_VEL
LIN {X 0,Y 479.924,Z 1012.685,A -85,B 0,C 180,E1 21862.943,E2 21862.943} C_VEL
LIN {X 0,Y 480.02,Z 1008.089,A -85,B 0,C 180,E1 21860.411,E2 21860.411} C_VEL
LIN {X 0,Y 480.217,Z 1002.445,A -85,B 0,C 180,E1 21857.986,E2 21857.986} C_VEL
LIN {X 0,Y 480.598,Z 994.163,A -85,B 0,C 180,E1 21855.177,E2 21855.177} C_VEL
LIN {X 0,Y 481.17,Z 984.935,A -85,B 0,C 180,E1 21852.593,E2 21852.593} C_VEL
LIN {X 0,Y 482.007,Z 973.742,A -85,B 0,C 180,E1 21849.989,E2 21849.989} C_VEL
LIN {X 0,Y 483.129,Z 961.275,A -85,B 0,C 180,E1 21847.493,E2 21847.493} C_VEL
LIN {X 0,Y 484.504,Z 947.37,A -85,B 0,C 180,E1 21845.107,E2 21845.107} C_VEL
LIN {X 0,Y 486.252,Z 931.215,A -85,B 0,C 180,E1 21842.711,E2 21842.711} C_VEL
LIN {X 0,Y 488.214,Z 914.567,A -85,B 0,C 180,E1 21840.564,E2 21840.564} C_VEL
LIN {X 0,Y 490.253,Z 896.82,A -85,B 0,C 180,E1 21838.6,E2 21838.6} C_VEL
LIN {X 0,Y 492.529,Z 877.682,A -85,B 0,C 180,E1 21836.759,E2 21836.759} C_VEL
LIN {X 0,Y 494.584,Z 859.378,A -85,B 0,C 180,E1 21835.248,E2 21835.248} C_VEL
LIN {X 0,Y 496.882,Z 837.898,A -85,B 0,C 180,E1 21833.734,E2 21833.734} C_VEL
LIN {X 0,Y 498.742,Z 818.542,A -85,B 0,C 180,E1 21832.601,E2 21832.601} C_VEL
LIN {X 0,Y 500.64,Z 795.735,A -85,B 0,C 180,E1 21831.499,E2 21831.499} C_VEL
LIN {X 0,Y 502.156,Z 774.437,A -85,B 0,C 180,E1 21830.679,E2 21830.679} C_VEL
LIN {X 0,Y 503.456,Z 751.473,A -85,B 0,C 180,E1 21830.016,E2 21830.016} C_VEL
LIN {X 0,Y 504.353,Z 728.559,A -85,B 0,C 180,E1 21829.546,E2 21829.546} C_VEL
LIN {X 0,Y 508.597,Z 522.414,A -85,B 0,C 180,E1 21826.117,E2 21826.117} C_VEL
LIN {X 0,Y 510.733,Z 421.002,A -85,B 0,C 180,E1 21824.382,E2 21824.382} C_VEL
LIN {X 0,Y 497.111,Z 399.914,A -85,B 0,C 180,E1 21822.321,E2 21822.321} C_VEL
LIN {X 0,Y 489.383,Z 388.502,A -85,B 0,C 180,E1 21821.06,E2 21821.06} C_VEL
LIN {X 0,Y 484.836,Z 379.599,A -85,B 0,C 180,E1 21819.586,E2 21819.586} C_VEL
LIN {X 0,Y 482.343,Z 374.9,A -85,B 0,C 180,E1 21818.757,E2 21818.757} C_VEL
LIN {X 0,Y 480.895,Z 371.305,A -85,B 0,C 180,E1 21818.096,E2 21818.096} C_VEL
LIN {X 0,Y 480.832,Z 371.118,A -85,B 0,C 180,E1 21814.576,E2 21814.576} C_VEL
LIN {X 0,Y 480.809,Z 371.128,A -85,B 0,C 180,E1 21811.185,E2 21811.185} C_VEL
LIN {X 0,Y 480.86,Z 371.15,A -85,B 0,C 180,E1 21807.759,E2 21807.759} C_VEL
LIN {X 0,Y 480.829,Z 371.155,A -85,B 0,C 180,E1 21804.313,E2 21804.313} C_VEL
LIN {X 0,Y 480.813,Z 371.152,A -85,B 0,C 180,E1 21800.83,E2 21800.83} C_VEL
LIN {X 0,Y 480.858,Z 371.144,A -85,B 0,C 180,E1 21797.385,E2 21797.385} C_VEL
LIN {X 0,Y 480.842,Z 371.145,A -85,B 0,C 180,E1 21793.958,E2 21793.958} C_VEL
LIN {X 0,Y 480.821,Z 371.149,A -85,B 0,C 180,E1 21790.421,E2 21790.421} C_VEL
LIN {X 0,Y 480.853,Z 371.15,A -85,B 0,C 180,E1 21786.926,E2 21786.926} C_VEL
LIN {X 0,Y 480.869,Z 371.146,A -85,B 0,C 180,E1 21783.457,E2 21783.457} C_VEL
LIN {X 0,Y 480.829,Z 371.15,A -85,B 0,C 180,E1 21780,E2 21780} C_VEL
LIN {X 0,Y 480.843,Z 371.15,A -85,B 0,C 180,E1 21776.389,E2 21776.389} C_VEL
LIN {X 0,Y 480.893,Z 371.148,A -85,B 0,C 180,E1 21772.833,E2 21772.833} C_VEL
LIN {X 0,Y 480.855,Z 371.148,A -85,B 0,C 180,E1 21769.335,E2 21769.335} C_VEL
LIN {X 0,Y 480.839,Z 371.149,A -85,B 0,C 180,E1 21765.796,E2 21765.796} C_VEL
LIN {X 0,Y 480.88,Z 371.147,A -85,B 0,C 180,E1 21762.328,E2 21762.328} C_VEL
LIN {X 0,Y 480.883,Z 371.145,A -85,B 0,C 180,E1 21758.79,E2 21758.79} C_VEL
LIN {X 0,Y 480.849,Z 371.146,A -85,B 0,C 180,E1 21755.294,E2 21755.294} C_VEL
LIN {X 0,Y 480.861,Z 371.146,A -85,B 0,C 180,E1 21751.7,E2 21751.7} C_VEL
LIN {X 0,Y 480.896,Z 371.146,A -85,B 0,C 180,E1 21748.243,E2 21748.243} C_VEL
LIN {X 0,Y 480.866,Z 371.147,A -85,B 0,C 180,E1 21744.687,E2 21744.687} C_VEL
LIN {X 0,Y 480.857,Z 371.148,A -85,B 0,C 180,E1 21741.04,E2 21741.04} C_VEL
LIN {X 0,Y 480.882,Z 371.145,A -85,B 0,C 180,E1 21737.487,E2 21737.487} C_VEL
LIN {X 0,Y 480.891,Z 371.143,A -85,B 0,C 180,E1 21733.977,E2 21733.977} C_VEL
LIN {X 0,Y 480.868,Z 371.145,A -85,B 0,C 180,E1 21730.44,E2 21730.44} C_VEL
LIN {X 0,Y 480.868,Z 371.142,A -85,B 0,C 180,E1 21726.781,E2 21726.781} C_VEL
LIN {X 0,Y 480.891,Z 371.146,A -85,B 0,C 180,E1 21723.144,E2 21723.144} C_VEL
LIN {X 0,Y 480.888,Z 371.124,A -85,B 0,C 180,E1 21719.518,E2 21719.518} C_VEL
LIN {X 0,Y 480.883,Z 371.15,A -85,B 0,C 180,E1 21717.945,E2 21717.945} C_VEL
LIN {X 0,Y 479.925,Z 371.275,A -85,B 0,C 180,E1 21717.027,E2 21717.027} C_VEL
LIN {X 0,Y 473.37,Z 372.075,A -85,B 0,C 180,E1 21714.379,E2 21714.379} C_VEL
LIN {X 0,Y 472.947,Z 372.133,A -85,B 0,C 180,E1 21713.772,E2 21713.772} C_VEL
LIN {X 0,Y 472.934,Z 372.117,A -85,B 0,C 180,E1 21710.154,E2 21710.154} C_VEL
LIN {X 0,Y 472.991,Z 372.445,A -85,B 0,C 180,E1 21709.122,E2 21709.122} C_VEL
LIN {X 0,Y 473.412,Z 373.992,A -85,B 0,C 180,E1 21708.881,E2 21708.881} C_VEL
LIN {X 0,Y 475.408,Z 376.961,A -85,B 0,C 180,E1 21708.512,E2 21708.512} C_VEL
LIN {X 0,Y 477.099,Z 378.534,A -85,B 0,C 180,E1 21708.23,E2 21708.23} C_VEL
LIN {X 0,Y 479.603,Z 382.34,A -85,B 0,C 180,E1 21707.783,E2 21707.783} C_VEL
LIN {X 0,Y 481.328,Z 384.318,A -85,B 0,C 180,E1 21707.495,E2 21707.495} C_VEL
LIN {X 0,Y 493.427,Z 400.865,A -85,B 0,C 180,E1 21705.52,E2 21705.52} C_VEL
LIN {X 0,Y 504.811,Z 417.137,A -85,B 0,C 180,E1 21703.792,E2 21703.792} C_VEL
LIN {X 0,Y 500.249,Z 609.764,A -85,B 0,C 180,E1 21700.498,E2 21700.498} C_VEL
LIN {X 0,Y 497.878,Z 712.208,A -85,B 0,C 180,E1 21698.761,E2 21698.761} C_VEL
LIN {X 0,Y 496.683,Z 735.019,A -85,B 0,C 180,E1 21698.181,E2 21698.181} C_VEL
LIN {X 0,Y 495.162,Z 757.03,A -85,B 0,C 180,E1 21697.422,E2 21697.422} C_VEL
LIN {X 0,Y 493.284,Z 778.74,A -85,B 0,C 180,E1 21696.456,E2 21696.456} C_VEL
LIN {X 0,Y 491.123,Z 800.572,A -85,B 0,C 180,E1 21695.253,E2 21695.253} C_VEL
LIN {X 0,Y 488.819,Z 821.325,A -85,B 0,C 180,E1 21693.867,E2 21693.867} C_VEL
LIN {X 0,Y 486.4,Z 841.259,A -85,B 0,C 180,E1 21692.294,E2 21692.294} C_VEL
LIN {X 0,Y 483.95,Z 861.023,A -85,B 0,C 180,E1 21690.464,E2 21690.464} C_VEL
LIN {X 0,Y 481.629,Z 879.198,A -85,B 0,C 180,E1 21688.51,E2 21688.51} C_VEL
LIN {X 0,Y 479.527,Z 896.087,A -85,B 0,C 180,E1 21686.411,E2 21686.411} C_VEL
LIN {X 0,Y 477.521,Z 912.611,A -85,B 0,C 180,E1 21684.035,E2 21684.035} C_VEL
LIN {X 0,Y 475.835,Z 927.529,A -85,B 0,C 180,E1 21681.539,E2 21681.539} C_VEL
LIN {X 0,Y 474.494,Z 940.868,A -85,B 0,C 180,E1 21678.942,E2 21678.942} C_VEL
LIN {X 0,Y 473.475,Z 952.527,A -85,B 0,C 180,E1 21676.266,E2 21676.266} C_VEL
LIN {X 0,Y 472.761,Z 962.561,A -85,B 0,C 180,E1 21673.534,E2 21673.534} C_VEL
LIN {X 0,Y 472.313,Z 970.689,A -85,B 0,C 180,E1 21670.842,E2 21670.842} C_VEL
LIN {X 0,Y 472.065,Z 977.329,A -85,B 0,C 180,E1 21668.081,E2 21668.081} C_VEL
LIN {X 0,Y 471.967,Z 982.181,A -85,B 0,C 180,E1 21665.464,E2 21665.464} C_VEL
LIN {X 0,Y 471.894,Z 985.756,A -85,B 0,C 180,E1 21662.597,E2 21662.597} C_VEL
LIN {X 0,Y 471.884,Z 987.532,A -85,B 0,C 180,E1 21659.994,E2 21659.994} C_VEL
LIN {X 0,Y 471.898,Z 987.896,A -85,B 0,C 180,E1 21657.264,E2 21657.264} C_VEL
LIN {X 0,Y 471.912,Z 986.754,A -85,B 0,C 180,E1 21654.509,E2 21654.509} C_VEL
LIN {X 0,Y 471.918,Z 984.044,A -85,B 0,C 180,E1 21651.779,E2 21651.779} C_VEL
LIN {X 0,Y 471.977,Z 980.165,A -85,B 0,C 180,E1 21649.269,E2 21649.269} C_VEL
LIN {X 0,Y 472.165,Z 974.365,A -85,B 0,C 180,E1 21646.508,E2 21646.508} C_VEL
LIN {X 0,Y 472.544,Z 966.588,A -85,B 0,C 180,E1 21643.642,E2 21643.642} C_VEL
LIN {X 0,Y 473.137,Z 957.121,A -85,B 0,C 180,E1 21640.837,E2 21640.837} C_VEL
LIN {X 0,Y 474.025,Z 946.073,A -85,B 0,C 180,E1 21638.113,E2 21638.113} C_VEL
LIN {X 0,Y 475.22,Z 933.488,A -85,B 0,C 180,E1 21635.485,E2 21635.485} C_VEL
LIN {X 0,Y 476.775,Z 918.985,A -85,B 0,C 180,E1 21632.899,E2 21632.899} C_VEL
LIN {X 0,Y 478.616,Z 903.392,A -85,B 0,C 180,E1 21630.507,E2 21630.507} C_VEL
LIN {X 0,Y 480.79,Z 886.044,A -85,B 0,C 180,E1 21628.213,E2 21628.213} C_VEL
LIN {X 0,Y 483.152,Z 867.303,A -85,B 0,C 180,E1 21626.082,E2 21626.082} C_VEL
LIN {X 0,Y 485.632,Z 847.836,A -85,B 0,C 180,E1 21624.187,E2 21624.187} C_VEL
LIN {X 0,Y 488.161,Z 827.01,A -85,B 0,C 180,E1 21622.458,E2 21622.458} C_VEL
LIN {X 0,Y 490.635,Z 805.413,A -85,B 0,C 180,E1 21620.956,E2 21620.956} C_VEL
LIN {X 0,Y 492.827,Z 783.912,A -85,B 0,C 180,E1 21619.713,E2 21619.713} C_VEL
LIN {X 0,Y 494.751,Z 761.656,A -85,B 0,C 180,E1 21618.676,E2 21618.676} C_VEL
LIN {X 0,Y 496.46,Z 738.195,A -85,B 0,C 180,E1 21617.83,E2 21617.83} C_VEL
LIN {X 0,Y 497.604,Z 717.403,A -85,B 0,C 180,E1 21617.271,E2 21617.271} C_VEL
LIN {X 0,Y 498.551,Z 685.433,A -85,B 0,C 180,E1 21616.683,E2 21616.683} C_VEL
LIN {X 0,Y 503.268,Z 480.289,A -85,B 0,C 180,E1 21613.216,E2 21613.216} C_VEL
LIN {X 0,Y 504.799,Z 417.039,A -85,B 0,C 180,E1 21612.106,E2 21612.106} C_VEL
LIN {X 0,Y 491.804,Z 398.372,A -85,B 0,C 180,E1 21610.07,E2 21610.07} C_VEL
LIN {X 0,Y 484.183,Z 388.125,A -85,B 0,C 180,E1 21608.79,E2 21608.79} C_VEL
LIN {X 0,Y 480.514,Z 383.201,A -85,B 0,C 180,E1 21608.135,E2 21608.135} C_VEL
LIN {X 0,Y 477.705,Z 379.572,A -85,B 0,C 180,E1 21607.623,E2 21607.623} C_VEL
LIN {X 0,Y 476.769,Z 378.012,A -85,B 0,C 180,E1 21607.441,E2 21607.441} C_VEL
LIN {X 0,Y 474.096,Z 375.379,A -85,B 0,C 180,E1 21606.95,E2 21606.95} C_VEL
LIN {X 0,Y 473.09,Z 372.974,A -85,B 0,C 180,E1 21606.676,E2 21606.676} C_VEL
LIN {X 0,Y 472.952,Z 372.158,A -85,B 0,C 180,E1 21606.312,E2 21606.312} C_VEL
LIN {X 0,Y 472.944,Z 372.133,A -85,B 0,C 180,E1 21602.666,E2 21602.666} C_VEL
LIN {X 0,Y 472.95,Z 372.136,A -85,B 0,C 180,E1 21599.031,E2 21599.031} C_VEL
LIN {X 0,Y 472.929,Z 372.129,A -85,B 0,C 180,E1 21595.392,E2 21595.392} C_VEL
LIN {X 0,Y 472.933,Z 372.135,A -85,B 0,C 180,E1 21591.735,E2 21591.735} C_VEL
LIN {X 0,Y 472.952,Z 372.137,A -85,B 0,C 180,E1 21588.167,E2 21588.167} C_VEL
LIN {X 0,Y 472.947,Z 372.134,A -85,B 0,C 180,E1 21584.552,E2 21584.552} C_VEL
LIN {X 0,Y 472.911,Z 372.138,A -85,B 0,C 180,E1 21580.999,E2 21580.999} C_VEL
LIN {X 0,Y 472.91,Z 372.141,A -85,B 0,C 180,E1 21577.369,E2 21577.369} C_VEL
LIN {X 0,Y 472.95,Z 372.136,A -85,B 0,C 180,E1 21573.914,E2 21573.914} C_VEL
LIN {X 0,Y 472.913,Z 372.131,A -85,B 0,C 180,E1 21570.348,E2 21570.348} C_VEL
LIN {X 0,Y 472.884,Z 372.146,A -85,B 0,C 180,E1 21566.796,E2 21566.796} C_VEL
LIN {X 0,Y 472.902,Z 372.182,A -85,B 0,C 180,E1 21563.249,E2 21563.249} C_VEL
LIN {X 0,Y 472.97,Z 372.711,A -85,B 0,C 180,E1 21562.909,E2 21562.909} C_VEL
LIN {X 0,Y 474.324,Z 375.815,A -85,B 0,C 180,E1 21562.316,E2 21562.316} C_VEL
LIN {X 0,Y 475.448,Z 377.381,A -85,B 0,C 180,E1 21561.963,E2 21561.963} C_VEL
LIN {X 0,Y 480.386,Z 386.948,A -85,B 0,C 180,E1 21560.265,E2 21560.265} C_VEL
LIN {X 0,Y 490.416,Z 401.789,A -85,B 0,C 180,E1 21558.501,E2 21558.501} C_VEL
LIN {X 0,Y 501.962,Z 419.712,A -85,B 0,C 180,E1 21556.65,E2 21556.65} C_VEL
LIN {X 0,Y 505.061,Z 425.059,A -85,B 0,C 180,E1 21556.171,E2 21556.171} C_VEL
LIN {X 0,Y 500.138,Z 630.864,A -85,B 0,C 180,E1 21552.653,E2 21552.653} C_VEL
LIN {X 0,Y 497.69,Z 739.98,A -85,B 0,C 180,E1 21550.815,E2 21550.815} C_VEL
LIN {X 0,Y 496.497,Z 762.734,A -85,B 0,C 180,E1 21550.247,E2 21550.247} C_VEL
LIN {X 0,Y 495.071,Z 784.289,A -85,B 0,C 180,E1 21549.524,E2 21549.524} C_VEL
LIN {X 0,Y 493.214,Z 806.379,A -85,B 0,C 180,E1 21548.565,E2 21548.565} C_VEL
LIN {X 0,Y 491.202,Z 827.99,A -85,B 0,C 180,E1 21547.419,E2 21547.419} C_VEL
LIN {X 0,Y 489.011,Z 848.669,A -85,B 0,C 180,E1 21546.078,E2 21546.078} C_VEL
LIN {X 0,Y 486.768,Z 868.509,A -85,B 0,C 180,E1 21544.575,E2 21544.575} C_VEL
LIN {X 0,Y 484.402,Z 887.234,A -85,B 0,C 180,E1 21542.881,E2 21542.881} C_VEL
LIN {X 0,Y 481.898,Z 907.03,A -85,B 0,C 180,E1 21540.798,E2 21540.798} C_VEL
LIN {X 0,Y 479.817,Z 923.638,A -85,B 0,C 180,E1 21538.777,E2 21538.777} C_VEL
LIN {X 0,Y 477.903,Z 939.12,A -85,B 0,C 180,E1 21536.6,E2 21536.6} C_VEL
LIN {X 0,Y 476.282,Z 953.49,A -85,B 0,C 180,E1 21534.299,E2 21534.299} C_VEL
LIN {X 0,Y 474.85,Z 966.914,A -85,B 0,C 180,E1 21531.786,E2 21531.786} C_VEL
LIN {X 0,Y 473.728,Z 979.281,A -85,B 0,C 180,E1 21529.098,E2 21529.098} C_VEL
LIN {X 0,Y 472.982,Z 989.055,A -85,B 0,C 180,E1 21526.584,E2 21526.584} C_VEL
LIN {X 0,Y 472.428,Z 998.3,A -85,B 0,C 180,E1 21523.729,E2 21523.729} C_VEL
LIN {X 0,Y 472.138,Z 1004.858,A -85,B 0,C 180,E1 21521.238,E2 21521.238} C_VEL
LIN {X 0,Y 471.994,Z 1010.643,A -85,B 0,C 180,E1 21518.4,E2 21518.4} C_VEL
LIN {X 0,Y 471.917,Z 1014.434,A -85,B 0,C 180,E1 21515.84,E2 21515.84} C_VEL
LIN {X 0,Y 471.887,Z 1016.984,A -85,B 0,C 180,E1 21513.04,E2 21513.04} C_VEL
LIN {X 0,Y 471.884,Z 1017.871,A -85,B 0,C 180,E1 21510.732,E2 21510.732} C_VEL
LIN {X 0,Y 471.909,Z 1017.596,A -85,B 0,C 180,E1 21508.061,E2 21508.061} C_VEL
LIN {X 0,Y 471.906,Z 1015.731,A -85,B 0,C 180,E1 21505.385,E2 21505.385} C_VEL
LIN {X 0,Y 471.932,Z 1012.5,A -85,B 0,C 180,E1 21502.7,E2 21502.7} C_VEL
LIN {X 0,Y 472.034,Z 1007.835,A -85,B 0,C 180,E1 21500.124,E2 21500.124} C_VEL
LIN {X 0,Y 472.28,Z 1001.836,A -85,B 0,C 180,E1 21497.533,E2 21497.533} C_VEL
LIN {X 0,Y 472.702,Z 993.757,A -85,B 0,C 180,E1 21494.798,E2 21494.798} C_VEL
LIN {X 0,Y 473.341,Z 984.46,A -85,B 0,C 180,E1 21492.168,E2 21492.168} C_VEL
LIN {X 0,Y 474.267,Z 973.167,A -85,B 0,C 180,E1 21489.519,E2 21489.519} C_VEL
LIN {X 0,Y 475.581,Z 959.872,A -85,B 0,C 180,E1 21486.854,E2 21486.854} C_VEL
LIN {X 0,Y 477.055,Z 946.597,A -85,B 0,C 180,E1 21484.559,E2 21484.559} C_VEL
LIN {X 0,Y 478.904,Z 930.751,A -85,B 0,C 180,E1 21482.189,E2 21482.189} C_VEL
LIN {X 0,Y 481.05,Z 913.926,A -85,B 0,C 180,E1 21480,E2 21480} C_VEL
LIN {X 0,Y 483.265,Z 896.21,A -85,B 0,C 180,E1 21478.023,E2 21478.023} C_VEL
LIN {X 0,Y 485.789,Z 876.297,A -85,B 0,C 180,E1 21476.103,E2 21476.103} C_VEL
LIN {X 0,Y 487.818,Z 859.294,A -85,B 0,C 180,E1 21474.695,E2 21474.695} C_VEL
LIN {X 0,Y 490.249,Z 837.476,A -85,B 0,C 180,E1 21473.163,E2 21473.163} C_VEL
LIN {X 0,Y 492.228,Z 818.044,A -85,B 0,C 180,E1 21472.019,E2 21472.019} C_VEL
LIN {X 0,Y 494.247,Z 795.151,A -85,B 0,C 180,E1 21470.906,E2 21470.906} C_VEL
LIN {X 0,Y 495.92,Z 773.406,A -85,B 0,C 180,E1 21470.068,E2 21470.068} C_VEL
LIN {X 0,Y 497.259,Z 751.051,A -85,B 0,C 180,E1 21469.424,E2 21469.424} C_VEL
LIN {X 0,Y 498.208,Z 728.117,A -85,B 0,C 180,E1 21468.95,E2 21468.95} C_VEL
LIN {X 0,Y 502.769,Z 523.011,A -85,B 0,C 180,E1 21465.5,E2 21465.5} C_VEL
LIN {X 0,Y 505.066,Z 424.574,A -85,B 0,C 180,E1 21463.799,E2 21463.799} C_VEL
LIN {X 0,Y 491.671,Z 403.917,A -85,B 0,C 180,E1 21461.72,E2 21461.72} C_VEL
LIN {X 0,Y 484.072,Z 393.014,A -85,B 0,C 180,E1 21460.472,E2 21460.472} C_VEL
LIN {X 0,Y 480.66,Z 387.876,A -85,B 0,C 180,E1 21459.843,E2 21459.843} C_VEL
LIN {X 0,Y 476.757,Z 380.336,A -85,B 0,C 180,E1 21458.526,E2 21458.526} C_VEL
LIN {X 0,Y 474.729,Z 376.304,A -85,B 0,C 180,E1 21457.799,E2 21457.799} C_VEL
LIN {X 0,Y 473.04,Z 373.037,A -85,B 0,C 180,E1 21457.177,E2 21457.177} C_VEL
LIN {X 0,Y 472.895,Z 372.252,A -85,B 0,C 180,E1 21456.953,E2 21456.953} C_VEL
LIN {X 0,Y 472.877,Z 372.132,A -85,B 0,C 180,E1 21453.349,E2 21453.349} C_VEL
LIN {X 0,Y 472.93,Z 372.099,A -85,B 0,C 180,E1 21449.92,E2 21449.92} C_VEL
LIN {X 0,Y 472.88,Z 372.138,A -85,B 0,C 180,E1 21446.496,E2 21446.496} C_VEL
LIN {X 0,Y 472.872,Z 372.135,A -85,B 0,C 180,E1 21442.895,E2 21442.895} C_VEL
LIN {X 0,Y 472.92,Z 372.136,A -85,B 0,C 180,E1 21439.464,E2 21439.464} C_VEL
LIN {X 0,Y 472.917,Z 372.14,A -85,B 0,C 180,E1 21435.869,E2 21435.869} C_VEL
LIN {X 0,Y 472.881,Z 372.142,A -85,B 0,C 180,E1 21432.377,E2 21432.377} C_VEL
LIN {X 0,Y 472.894,Z 372.137,A -85,B 0,C 180,E1 21428.756,E2 21428.756} C_VEL
LIN {X 0,Y 472.942,Z 372.131,A -85,B 0,C 180,E1 21425.337,E2 21425.337} C_VEL
LIN {X 0,Y 472.9,Z 372.138,A -85,B 0,C 180,E1 21421.817,E2 21421.817} C_VEL
LIN {X 0,Y 472.895,Z 372.135,A -85,B 0,C 180,E1 21418.303,E2 21418.303} C_VEL
LIN {X 0,Y 472.94,Z 372.128,A -85,B 0,C 180,E1 21414.784,E2 21414.784} C_VEL
LIN {X 0,Y 472.926,Z 372.134,A -85,B 0,C 180,E1 21411.244,E2 21411.244} C_VEL
LIN {X 0,Y 472.901,Z 372.137,A -85,B 0,C 180,E1 21407.669,E2 21407.669} C_VEL
LIN {X 0,Y 472.914,Z 372.131,A -85,B 0,C 180,E1 21404.046,E2 21404.046} C_VEL
LIN {X 0,Y 472.952,Z 372.127,A -85,B 0,C 180,E1 21400.486,E2 21400.486} C_VEL
LIN {X 0,Y 472.925,Z 372.134,A -85,B 0,C 180,E1 21396.975,E2 21396.975} C_VEL
LIN {X 0,Y 472.912,Z 372.135,A -85,B 0,C 180,E1 21393.37,E2 21393.37} C_VEL
LIN {X 0,Y 472.933,Z 372.128,A -85,B 0,C 180,E1 21389.79,E2 21389.79} C_VEL
LIN {X 0,Y 472.955,Z 372.127,A -85,B 0,C 180,E1 21386.175,E2 21386.175} C_VEL
LIN {X 0,Y 472.927,Z 372.132,A -85,B 0,C 180,E1 21382.641,E2 21382.641} C_VEL
LIN {X 0,Y 472.92,Z 372.128,A -85,B 0,C 180,E1 21378.999,E2 21378.999} C_VEL
LIN {X 0,Y 472.945,Z 372.133,A -85,B 0,C 180,E1 21375.421,E2 21375.421} C_VEL
LIN {X 0,Y 472.954,Z 372.136,A -85,B 0,C 180,E1 21371.731,E2 21371.731} C_VEL
LIN {X 0,Y 472.944,Z 372.135,A -85,B 0,C 180,E1 21368.115,E2 21368.115} C_VEL
LIN {X 0,Y 472.928,Z 372.131,A -85,B 0,C 180,E1 21364.458,E2 21364.458} C_VEL
LIN {X 0,Y 472.937,Z 372.105,A -85,B 0,C 180,E1 21360.767,E2 21360.767} C_VEL
LIN {X 0,Y 472.95,Z 372.125,A -85,B 0,C 180,E1 21357.122,E2 21357.122} C_VEL
LIN {X 0,Y 472.947,Z 372.133,A -85,B 0,C 180,E1 21353.772,E2 21353.772} C_VEL
LIN {X 0,Y 471.956,Z 372.259,A -85,B 0,C 180,E1 21353.152,E2 21353.152} C_VEL
LIN {X 0,Y 465.545,Z 373.027,A -85,B 0,C 180,E1 21351.466,E2 21351.466} C_VEL
LIN {X 0,Y 465.003,Z 373.093,A -85,B 0,C 180,E1 21351.008,E2 21351.008} C_VEL
LIN {X 0,Y 465.018,Z 373.239,A -85,B 0,C 180,E1 21350.369,E2 21350.369} C_VEL
LIN {X 0,Y 465.354,Z 374.676,A -85,B 0,C 180,E1 21350.087,E2 21350.087} C_VEL
LIN {X 0,Y 467.296,Z 377.79,A -85,B 0,C 180,E1 21349.702,E2 21349.702} C_VEL
LIN {X 0,Y 469.226,Z 379.541,A -85,B 0,C 180,E1 21349.367,E2 21349.367} C_VEL
LIN {X 0,Y 471.8,Z 383.428,A -85,B 0,C 180,E1 21348.89,E2 21348.89} C_VEL
LIN {X 0,Y 473.609,Z 385.449,A -85,B 0,C 180,E1 21348.574,E2 21348.574} C_VEL
LIN {X 0,Y 476.984,Z 389.83,A -85,B 0,C 180,E1 21347.981,E2 21347.981} C_VEL
LIN {X 0,Y 491.755,Z 410.164,A -85,B 0,C 180,E1 21345.532,E2 21345.532} C_VEL
LIN {X 0,Y 499.194,Z 421.34,A -85,B 0,C 180,E1 21344.373,E2 21344.373} C_VEL
LIN {X 0,Y 493.761,Z 634.122,A -85,B 0,C 180,E1 21340.711,E2 21340.711} C_VEL
LIN {X 0,Y 491.762,Z 713.081,A -85,B 0,C 180,E1 21339.35,E2 21339.35} C_VEL
LIN {X 0,Y 490.494,Z 735.544,A -85,B 0,C 180,E1 21338.769,E2 21338.769} C_VEL
LIN {X 0,Y 488.889,Z 757.666,A -85,B 0,C 180,E1 21337.998,E2 21337.998} C_VEL
LIN {X 0,Y 486.879,Z 779.443,A -85,B 0,C 180,E1 21337.015,E2 21337.015} C_VEL
LIN {X 0,Y 484.489,Z 802.233,A -85,B 0,C 180,E1 21335.741,E2 21335.741} C_VEL
LIN {X 0,Y 482.041,Z 822.784,A -85,B 0,C 180,E1 21334.339,E2 21334.339} C_VEL
LIN {X 0,Y 479.375,Z 843.215,A -85,B 0,C 180,E1 21332.687,E2 21332.687} C_VEL
LIN {X 0,Y 476.615,Z 863.813,A -85,B 0,C 180,E1 21330.718,E2 21330.718} C_VEL
LIN {X 0,Y 474.065,Z 882.187,A -85,B 0,C 180,E1 21328.662,E2 21328.662} C_VEL
LIN {X 0,Y 471.669,Z 899.969,A -85,B 0,C 180,E1 21326.351,E2 21326.351} C_VEL
LIN {X 0,Y 469.566,Z 916.27,A -85,B 0,C 180,E1 21323.885,E2 21323.885} C_VEL
LIN {X 0,Y 467.79,Z 931.12,A -85,B 0,C 180,E1 21321.268,E2 21321.268} C_VEL
LIN {X 0,Y 466.421,Z 943.947,A -85,B 0,C 180,E1 21318.623,E2 21318.623} C_VEL
LIN {X 0,Y 465.421,Z 954.993,A -85,B 0,C 180,E1 21315.948,E2 21315.948} C_VEL
LIN {X 0,Y 464.727,Z 964.468,A -85,B 0,C 180,E1 21313.22,E2 21313.22} C_VEL
LIN {X 0,Y 464.274,Z 972.534,A -85,B 0,C 180,E1 21310.366,E2 21310.366} C_VEL
LIN {X 0,Y 464.054,Z 978.439,A -85,B 0,C 180,E1 21307.712,E2 21307.712} C_VEL
LIN {X 0,Y 463.947,Z 983.231,A -85,B 0,C 180,E1 21304.844,E2 21304.844} C_VEL
LIN {X 0,Y 463.905,Z 986.354,A -85,B 0,C 180,E1 21301.972,E2 21301.972} C_VEL
LIN {X 0,Y 463.909,Z 987.792,A -85,B 0,C 180,E1 21299.28,E2 21299.28} C_VEL
LIN {X 0,Y 463.905,Z 987.798,A -85,B 0,C 180,E1 21296.658,E2 21296.658} C_VEL
LIN {X 0,Y 463.904,Z 986.346,A -85,B 0,C 180,E1 21293.925,E2 21293.925} C_VEL
LIN {X 0,Y 463.945,Z 983.249,A -85,B 0,C 180,E1 21291.078,E2 21291.078} C_VEL
LIN {X 0,Y 464.058,Z 978.447,A -85,B 0,C 180,E1 21288.202,E2 21288.202} C_VEL
LIN {X 0,Y 464.29,Z 972.197,A -85,B 0,C 180,E1 21285.406,E2 21285.406} C_VEL
LIN {X 0,Y 464.742,Z 964.253,A -85,B 0,C 180,E1 21282.624,E2 21282.624} C_VEL
LIN {X 0,Y 465.435,Z 954.84,A -85,B 0,C 180,E1 21279.92,E2 21279.92} C_VEL
LIN {X 0,Y 466.463,Z 943.526,A -85,B 0,C 180,E1 21277.191,E2 21277.191} C_VEL
LIN {X 0,Y 467.801,Z 931.023,A -85,B 0,C 180,E1 21274.623,E2 21274.623} C_VEL
LIN {X 0,Y 469.572,Z 916.237,A -85,B 0,C 180,E1 21272.019,E2 21272.019} C_VEL
LIN {X 0,Y 471.627,Z 900.275,A -85,B 0,C 180,E1 21269.602,E2 21269.602} C_VEL
LIN {X 0,Y 473.949,Z 883.075,A -85,B 0,C 180,E1 21267.355,E2 21267.355} C_VEL
LIN {X 0,Y 476.595,Z 863.956,A -85,B 0,C 180,E1 21265.207,E2 21265.207} C_VEL
LIN {X 0,Y 479.278,Z 843.968,A -85,B 0,C 180,E1 21263.287,E2 21263.287} C_VEL
LIN {X 0,Y 481.994,Z 823.293,A -85,B 0,C 180,E1 21261.606,E2 21261.606} C_VEL
LIN {X 0,Y 484.391,Z 803.165,A -85,B 0,C 180,E1 21260.228,E2 21260.228} C_VEL
LIN {X 0,Y 486.783,Z 780.295,A -85,B 0,C 180,E1 21258.938,E2 21258.938} C_VEL
LIN {X 0,Y 488.834,Z 758.224,A -85,B 0,C 180,E1 21257.935,E2 21257.935} C_VEL
LIN {X 0,Y 490.391,Z 736.492,A -85,B 0,C 180,E1 21257.177,E2 21257.177} C_VEL
LIN {X 0,Y 491.619,Z 715.202,A -85,B 0,C 180,E1 21256.614,E2 21256.614} C_VEL
LIN {X 0,Y 492.802,Z 671.815,A -85,B 0,C 180,E1 21255.846,E2 21255.846} C_VEL
LIN {X 0,Y 497.934,Z 468.382,A -85,B 0,C 180,E1 21252.356,E2 21252.356} C_VEL
LIN {X 0,Y 499.137,Z 420.87,A -85,B 0,C 180,E1 21251.497,E2 21251.497} C_VEL
LIN {X 0,Y 487.642,Z 404.26,A -85,B 0,C 180,E1 21249.65,E2 21249.65} C_VEL
LIN {X 0,Y 479.88,Z 393.747,A -85,B 0,C 180,E1 21248.299,E2 21248.299} C_VEL
LIN {X 0,Y 476.688,Z 389.452,A -85,B 0,C 180,E1 21247.715,E2 21247.715} C_VEL
LIN {X 0,Y 473,Z 384.495,A -85,B 0,C 180,E1 21247.012,E2 21247.012} C_VEL
LIN {X 0,Y 470.126,Z 381.014,A -85,B 0,C 180,E1 21246.453,E2 21246.453} C_VEL
LIN {X 0,Y 468.966,Z 379.074,A -85,B 0,C 180,E1 21246.209,E2 21246.209} C_VEL
LIN {X 0,Y 466.231,Z 376.49,A -85,B 0,C 180,E1 21245.677,E2 21245.677} C_VEL
LIN {X 0,Y 465.156,Z 373.954,A -85,B 0,C 180,E1 21245.366,E2 21245.366} C_VEL
LIN {X 0,Y 465.014,Z 373.169,A -85,B 0,C 180,E1 21245.058,E2 21245.058} C_VEL
LIN {X 0,Y 465.003,Z 373.126,A -85,B 0,C 180,E1 21241.356,E2 21241.356} C_VEL
LIN {X 0,Y 464.994,Z 373.119,A -85,B 0,C 180,E1 21237.659,E2 21237.659} C_VEL
LIN {X 0,Y 465.007,Z 373.126,A -85,B 0,C 180,E1 21233.953,E2 21233.953} C_VEL
LIN {X 0,Y 465.013,Z 373.124,A -85,B 0,C 180,E1 21230.221,E2 21230.221} C_VEL
LIN {X 0,Y 465.009,Z 373.125,A -85,B 0,C 180,E1 21226.573,E2 21226.573} C_VEL
LIN {X 0,Y 464.976,Z 373.129,A -85,B 0,C 180,E1 21222.996,E2 21222.996} C_VEL
LIN {X 0,Y 464.972,Z 373.129,A -85,B 0,C 180,E1 21219.298,E2 21219.298} C_VEL
LIN {X 0,Y 464.998,Z 373.119,A -85,B 0,C 180,E1 21215.745,E2 21215.745} C_VEL
LIN {X 0,Y 465.011,Z 373.125,A -85,B 0,C 180,E1 21212.048,E2 21212.048} C_VEL
LIN {X 0,Y 464.954,Z 373.128,A -85,B 0,C 180,E1 21208.622,E2 21208.622} C_VEL
LIN {X 0,Y 464.945,Z 373.127,A -85,B 0,C 180,E1 21204.958,E2 21204.958} C_VEL
LIN {X 0,Y 465.037,Z 373.578,A -85,B 0,C 180,E1 21204.155,E2 21204.155} C_VEL
LIN {X 0,Y 466.603,Z 377.054,A -85,B 0,C 180,E1 21203.437,E2 21203.437} C_VEL
LIN {X 0,Y 467.63,Z 378.706,A -85,B 0,C 180,E1 21203.072,E2 21203.072} C_VEL
LIN {X 0,Y 469.589,Z 382.354,A -85,B 0,C 180,E1 21202.332,E2 21202.332} C_VEL
LIN {X 0,Y 471.855,Z 386.558,A -85,B 0,C 180,E1 21201.583,E2 21201.583} C_VEL
LIN {X 0,Y 479.69,Z 397.671,A -85,B 0,C 180,E1 21200.099,E2 21200.099} C_VEL
LIN {X 0,Y 489.985,Z 413.203,A -85,B 0,C 180,E1 21198.3,E2 21198.3} C_VEL
LIN {X 0,Y 499.408,Z 428.647,A -85,B 0,C 180,E1 21196.771,E2 21196.771} C_VEL
LIN {X 0,Y 494.135,Z 632.455,A -85,B 0,C 180,E1 21193.245,E2 21193.245} C_VEL
LIN {X 0,Y 491.528,Z 739.769,A -85,B 0,C 180,E1 21191.413,E2 21191.413} C_VEL
LIN {X 0,Y 490.236,Z 762.739,A -85,B 0,C 180,E1 21190.834,E2 21190.834} C_VEL
LIN {X 0,Y 488.653,Z 785.197,A -85,B 0,C 180,E1 21190.07,E2 21190.07} C_VEL
LIN {X 0,Y 486.677,Z 806.951,A -85,B 0,C 180,E1 21189.105,E2 21189.105} C_VEL
LIN {X 0,Y 484.525,Z 828.368,A -85,B 0,C 180,E1 21187.951,E2 21187.951} C_VEL
LIN {X 0,Y 482.203,Z 848.87,A -85,B 0,C 180,E1 21186.603,E2 21186.603} C_VEL
LIN {X 0,Y 479.666,Z 869.905,A -85,B 0,C 180,E1 21184.978,E2 21184.978} C_VEL
LIN {X 0,Y 477.282,Z 888.531,A -85,B 0,C 180,E1 21183.292,E2 21183.292} C_VEL
LIN {X 0,Y 474.728,Z 907.371,A -85,B 0,C 180,E1 21181.272,E2 21181.272} C_VEL
LIN {X 0,Y 472.459,Z 924.143,A -85,B 0,C 180,E1 21179.199,E2 21179.199} C_VEL
LIN {X 0,Y 470.353,Z 939.964,A -85,B 0,C 180,E1 21176.925,E2 21176.925} C_VEL
LIN {X 0,Y 468.521,Z 954.927,A -85,B 0,C 180,E1 21174.46,E2 21174.46} C_VEL
LIN {X 0,Y 467.057,Z 967.701,A -85,B 0,C 180,E1 21172.004,E2 21172.004} C_VEL
LIN {X 0,Y 465.817,Z 980.312,A -85,B 0,C 180,E1 21169.175,E2 21169.175} C_VEL
LIN {X 0,Y 465.005,Z 990.43,A -85,B 0,C 180,E1 21166.492,E2 21166.492} C_VEL
LIN {X 0,Y 464.463,Z 998.692,A -85,B 0,C 180,E1 21163.828,E2 21163.828} C_VEL
LIN {X 0,Y 464.147,Z 1005.463,A -85,B 0,C 180,E1 21161.182,E2 21161.182} C_VEL
LIN {X 0,Y 463.998,Z 1010.837,A -85,B 0,C 180,E1 21158.429,E2 21158.429} C_VEL
LIN {X 0,Y 463.918,Z 1014.593,A -85,B 0,C 180,E1 21155.817,E2 21155.817} C_VEL
LIN {X 0,Y 463.886,Z 1016.984,A -85,B 0,C 180,E1 21153.092,E2 21153.092} C_VEL
LIN {X 0,Y 463.885,Z 1017.871,A -85,B 0,C 180,E1 21150.744,E2 21150.744} C_VEL
LIN {X 0,Y 463.91,Z 1017.596,A -85,B 0,C 180,E1 21148.027,E2 21148.027} C_VEL
LIN {X 0,Y 463.907,Z 1015.845,A -85,B 0,C 180,E1 21145.429,E2 21145.429} C_VEL
LIN {X 0,Y 463.934,Z 1012.685,A -85,B 0,C 180,E1 21142.698,E2 21142.698} C_VEL
LIN {X 0,Y 464.044,Z 1008.089,A -85,B 0,C 180,E1 21140.078,E2 21140.078} C_VEL
LIN {X 0,Y 464.305,Z 1002.141,A -85,B 0,C 180,E1 21137.442,E2 21137.442} C_VEL
LIN {X 0,Y 464.76,Z 994.161,A -85,B 0,C 180,E1 21134.66,E2 21134.66} C_VEL
LIN {X 0,Y 465.446,Z 984.938,A -85,B 0,C 180,E1 21131.985,E2 21131.985} C_VEL
LIN {X 0,Y 466.444,Z 973.739,A -85,B 0,C 180,E1 21129.291,E2 21129.291} C_VEL
LIN {X 0,Y 467.789,Z 961.272,A -85,B 0,C 180,E1 21126.712,E2 21126.712} C_VEL
LIN {X 0,Y 469.407,Z 947.597,A -85,B 0,C 180,E1 21124.29,E2 21124.29} C_VEL
LIN {X 0,Y 471.49,Z 931.212,A -85,B 0,C 180,E1 21121.782,E2 21121.782} C_VEL
LIN {X 0,Y 473.771,Z 914.566,A -85,B 0,C 180,E1 21119.574,E2 21119.574} C_VEL
LIN {X 0,Y 476.13,Z 897.052,A -85,B 0,C 180,E1 21117.584,E2 21117.584} C_VEL
LIN {X 0,Y 478.468,Z 879.768,A -85,B 0,C 180,E1 21115.874,E2 21115.874} C_VEL
LIN {X 0,Y 480.846,Z 860.499,A -85,B 0,C 180,E1 21114.251,E2 21114.251} C_VEL
LIN {X 0,Y 483.325,Z 840.057,A -85,B 0,C 180,E1 21112.77,E2 21112.77} C_VEL
LIN {X 0,Y 485.52,Z 819.835,A -85,B 0,C 180,E1 21111.549,E2 21111.549} C_VEL
LIN {X 0,Y 487.598,Z 798.754,A -85,B 0,C 180,E1 21110.481,E2 21110.481} C_VEL
LIN {X 0,Y 489.381,Z 776.74,A -85,B 0,C 180,E1 21109.597,E2 21109.597} C_VEL
LIN {X 0,Y 491.018,Z 752.43,A -85,B 0,C 180,E1 21108.86,E2 21108.86} C_VEL
LIN {X 0,Y 492.002,Z 730.785,A -85,B 0,C 180,E1 21108.398,E2 21108.398} C_VEL
LIN {X 0,Y 497.045,Z 521.845,A -85,B 0,C 180,E1 21104.838,E2 21104.838} C_VEL
LIN {X 0,Y 499.38,Z 428.2,A -85,B 0,C 180,E1 21103.196,E2 21103.196} C_VEL
LIN {X 0,Y 487.154,Z 409.29,A -85,B 0,C 180,E1 21101.25,E2 21101.25} C_VEL
LIN {X 0,Y 475.277,Z 391.938,A -85,B 0,C 180,E1 21099.21,E2 21099.21} C_VEL
LIN {X 0,Y 472.266,Z 387.665,A -85,B 0,C 180,E1 21098.634,E2 21098.634} C_VEL
LIN {X 0,Y 469.111,Z 381.77,A -85,B 0,C 180,E1 21097.553,E2 21097.553} C_VEL
LIN {X 0,Y 466.744,Z 377.269,A -85,B 0,C 180,E1 21096.703,E2 21096.703} C_VEL
LIN {X 0,Y 465.027,Z 373.433,A -85,B 0,C 180,E1 21095.942,E2 21095.942} C_VEL
LIN {X 0,Y 464.975,Z 373.092,A -85,B 0,C 180,E1 21094.346,E2 21094.346} C_VEL
LIN {X 0,Y 464.931,Z 373.096,A -85,B 0,C 180,E1 21090.909,E2 21090.909} C_VEL
LIN {X 0,Y 464.94,Z 373.133,A -85,B 0,C 180,E1 21087.261,E2 21087.261} C_VEL
LIN {X 0,Y 464.984,Z 373.12,A -85,B 0,C 180,E1 21083.66,E2 21083.66} C_VEL
LIN {X 0,Y 464.961,Z 373.123,A -85,B 0,C 180,E1 21080.124,E2 21080.124} C_VEL
LIN {X 0,Y 464.938,Z 373.128,A -85,B 0,C 180,E1 21076.619,E2 21076.619} C_VEL
LIN {X 0,Y 464.967,Z 373.131,A -85,B 0,C 180,E1 21073.086,E2 21073.086} C_VEL
LIN {X 0,Y 464.995,Z 373.129,A -85,B 0,C 180,E1 21069.53,E2 21069.53} C_VEL
LIN {X 0,Y 464.952,Z 373.13,A -85,B 0,C 180,E1 21066.048,E2 21066.048} C_VEL
LIN {X 0,Y 464.952,Z 373.128,A -85,B 0,C 180,E1 21062.341,E2 21062.341} C_VEL
LIN {X 0,Y 464.99,Z 373.122,A -85,B 0,C 180,E1 21058.815,E2 21058.815} C_VEL
LIN {X 0,Y 464.999,Z 373.122,A -85,B 0,C 180,E1 21055.189,E2 21055.189} C_VEL
LIN {X 0,Y 464.962,Z 373.129,A -85,B 0,C 180,E1 21051.716,E2 21051.716} C_VEL
LIN {X 0,Y 464.964,Z 373.125,A -85,B 0,C 180,E1 21047.96,E2 21047.96} C_VEL
LIN {X 0,Y 465.002,Z 373.119,A -85,B 0,C 180,E1 21044.408,E2 21044.408} C_VEL
LIN {X 0,Y 465.006,Z 373.12,A -85,B 0,C 180,E1 21040.793,E2 21040.793} C_VEL
LIN {X 0,Y 464.974,Z 373.128,A -85,B 0,C 180,E1 21037.228,E2 21037.228} C_VEL
LIN {X 0,Y 464.975,Z 373.123,A -85,B 0,C 180,E1 21033.568,E2 21033.568} C_VEL
LIN {X 0,Y 465.018,Z 373.115,A -85,B 0,C 180,E1 21030.046,E2 21030.046} C_VEL
LIN {X 0,Y 465.007,Z 373.119,A -85,B 0,C 180,E1 21026.454,E2 21026.454} C_VEL
LIN {X 0,Y 464.98,Z 373.121,A -85,B 0,C 180,E1 21022.825,E2 21022.825} C_VEL
LIN {X 0,Y 464.984,Z 373.116,A -85,B 0,C 180,E1 21019.179,E2 21019.179} C_VEL
LIN {X 0,Y 465.01,Z 373.12,A -85,B 0,C 180,E1 21015.543,E2 21015.543} C_VEL
LIN {X 0,Y 465.013,Z 373.124,A -85,B 0,C 180,E1 21011.93,E2 21011.93} C_VEL
LIN {X 0,Y 464.999,Z 373.127,A -85,B 0,C 180,E1 21008.257,E2 21008.257} C_VEL
LIN {X 0,Y 464.989,Z 373.12,A -85,B 0,C 180,E1 21004.557,E2 21004.557} C_VEL
LIN {X 0,Y 465.006,Z 373.092,A -85,B 0,C 180,E1 21000.914,E2 21000.914} C_VEL
LIN {X 0,Y 465.009,Z 373.115,A -85,B 0,C 180,E1 20997.253,E2 20997.253} C_VEL
LIN {X 0,Y 465.013,Z 373.125,A -85,B 0,C 180,E1 20993.569,E2 20993.569} C_VEL
LIN {X 0,Y 465.003,Z 373.093,A -85,B 0,C 180,E1 20991.008,E2 20991.008} C_VEL
LIN {X 0,Y 465.056,Z 374.204,A -85,B 0,C 180,E1 20990.593,E2 20990.593} C_VEL
LIN {X 0,Y 465.253,Z 377.312,A -85,B 0,C 180,E1 20990.199,E2 20990.199} C_VEL
LIN {X 0,Y 466.386,Z 384.924,A -85,B 0,C 180,E1 20989.667,E2 20989.667} C_VEL
LIN {X 0,Y 468.078,Z 389.458,A -85,B 0,C 180,E1 20989.296,E2 20989.296} C_VEL
LIN {X 0,Y 469.173,Z 390.881,A -85,B 0,C 180,E1 20989.098,E2 20989.098} C_VEL
LIN {X 0,Y 481.651,Z 407.765,A -85,B 0,C 180,E1 20986.916,E2 20986.916} C_VEL
LIN {X 0,Y 493.588,Z 424.858,A -85,B 0,C 180,E1 20984.987,E2 20984.987} C_VEL
LIN {X 0,Y 487.791,Z 637.089,A -85,B 0,C 180,E1 20981.296,E2 20981.296} C_VEL
LIN {X 0,Y 485.724,Z 713.227,A -85,B 0,C 180,E1 20979.969,E2 20979.969} C_VEL
LIN {X 0,Y 484.393,Z 735.55,A -85,B 0,C 180,E1 20979.387,E2 20979.387} C_VEL
LIN {X 0,Y 482.747,Z 757.398,A -85,B 0,C 180,E1 20978.625,E2 20978.625} C_VEL
LIN {X 0,Y 480.644,Z 778.979,A -85,B 0,C 180,E1 20977.647,E2 20977.647} C_VEL
LIN {X 0,Y 478.208,Z 801.039,A -85,B 0,C 180,E1 20976.419,E2 20976.419} C_VEL
LIN {X 0,Y 475.607,Z 821.823,A -85,B 0,C 180,E1 20975.003,E2 20975.003} C_VEL
LIN {X 0,Y 472.664,Z 843.153,A -85,B 0,C 180,E1 20973.271,E2 20973.271} C_VEL
LIN {X 0,Y 469.775,Z 863.204,A -85,B 0,C 180,E1 20971.338,E2 20971.338} C_VEL
LIN {X 0,Y 466.886,Z 882.612,A -85,B 0,C 180,E1 20969.138,E2 20969.138} C_VEL
LIN {X 0,Y 464.306,Z 900.337,A -85,B 0,C 180,E1 20966.787,E2 20966.787} C_VEL
LIN {X 0,Y 462.037,Z 916.591,A -85,B 0,C 180,E1 20964.284,E2 20964.284} C_VEL
LIN {X 0,Y 460.122,Z 931.391,A -85,B 0,C 180,E1 20961.625,E2 20961.625} C_VEL
LIN {X 0,Y 458.599,Z 944.562,A -85,B 0,C 180,E1 20958.847,E2 20958.847} C_VEL
LIN {X 0,Y 457.472,Z 956.12,A -85,B 0,C 180,E1 20955.957,E2 20955.957} C_VEL
LIN {X 0,Y 456.751,Z 965.327,A -85,B 0,C 180,E1 20953.202,E2 20953.202} C_VEL
LIN {X 0,Y 456.292,Z 972.959,A -85,B 0,C 180,E1 20950.409,E2 20950.409} C_VEL
LIN {X 0,Y 456.059,Z 979.066,A -85,B 0,C 180,E1 20947.572,E2 20947.572} C_VEL
LIN {X 0,Y 455.945,Z 983.622,A -85,B 0,C 180,E1 20944.681,E2 20944.681} C_VEL
LIN {X 0,Y 455.911,Z 986.506,A -85,B 0,C 180,E1 20941.84,E2 20941.84} C_VEL
LIN {X 0,Y 455.913,Z 987.849,A -85,B 0,C 180,E1 20938.975,E2 20938.975} C_VEL
LIN {X 0,Y 455.887,Z 987.705,A -85,B 0,C 180,E1 20936.226,E2 20936.226} C_VEL
LIN {X 0,Y 455.891,Z 986.098,A -85,B 0,C 180,E1 20933.531,E2 20933.531} C_VEL
LIN {X 0,Y 455.964,Z 982.854,A -85,B 0,C 180,E1 20930.671,E2 20930.671} C_VEL
LIN {X 0,Y 456.08,Z 978.024,A -85,B 0,C 180,E1 20927.817,E2 20927.817} C_VEL
LIN {X 0,Y 456.349,Z 971.839,A -85,B 0,C 180,E1 20925.048,E2 20925.048} C_VEL
LIN {X 0,Y 456.864,Z 963.817,A -85,B 0,C 180,E1 20922.213,E2 20922.213} C_VEL
LIN {X 0,Y 457.706,Z 953.78,A -85,B 0,C 180,E1 20919.31,E2 20919.31} C_VEL
LIN {X 0,Y 458.903,Z 942.042,A -85,B 0,C 180,E1 20916.486,E2 20916.486} C_VEL
LIN {X 0,Y 460.499,Z 928.562,A -85,B 0,C 180,E1 20913.735,E2 20913.735} C_VEL
LIN {X 0,Y 462.465,Z 913.481,A -85,B 0,C 180,E1 20911.109,E2 20911.109} C_VEL
LIN {X 0,Y 464.767,Z 897.15,A -85,B 0,C 180,E1 20908.669,E2 20908.669} C_VEL
LIN {X 0,Y 467.518,Z 878.547,A -85,B 0,C 180,E1 20906.277,E2 20906.277} C_VEL
LIN {X 0,Y 470.375,Z 859.258,A -85,B 0,C 180,E1 20904.154,E2 20904.154} C_VEL
LIN {X 0,Y 473.159,Z 840.008,A -85,B 0,C 180,E1 20902.357,E2 20902.357} C_VEL
LIN {X 0,Y 475.859,Z 819.942,A -85,B 0,C 180,E1 20900.766,E2 20900.766} C_VEL
LIN {X 0,Y 478.509,Z 798.652,A -85,B 0,C 180,E1 20899.341,E2 20899.341} C_VEL
LIN {X 0,Y 480.752,Z 777.894,A -85,B 0,C 180,E1 20898.21,E2 20898.21} C_VEL
LIN {X 0,Y 482.871,Z 755.381,A -85,B 0,C 180,E1 20897.212,E2 20897.212} C_VEL
LIN {X 0,Y 484.395,Z 734.827,A -85,B 0,C 180,E1 20896.508,E2 20896.508} C_VEL
LIN {X 0,Y 485.695,Z 711.587,A -85,B 0,C 180,E1 20895.92,E2 20895.92} C_VEL
LIN {X 0,Y 491.515,Z 497.491,A -85,B 0,C 180,E1 20892.199,E2 20892.199} C_VEL
LIN {X 0,Y 493.615,Z 424.663,A -85,B 0,C 180,E1 20890.888,E2 20890.888} C_VEL
LIN {X 0,Y 480.929,Z 406.371,A -85,B 0,C 180,E1 20888.76,E2 20888.76} C_VEL
LIN {X 0,Y 472.91,Z 395.654,A -85,B 0,C 180,E1 20887.288,E2 20887.288} C_VEL
LIN {X 0,Y 469.288,Z 390.832,A -85,B 0,C 180,E1 20886.576,E2 20886.576} C_VEL
LIN {X 0,Y 466.097,Z 386.452,A -85,B 0,C 180,E1 20885.926,E2 20885.926} C_VEL
LIN {X 0,Y 462.595,Z 382.527,A -85,B 0,C 180,E1 20885.209,E2 20885.209} C_VEL
LIN {X 0,Y 461.324,Z 380.237,A -85,B 0,C 180,E1 20884.912,E2 20884.912} C_VEL
LIN {X 0,Y 458.5,Z 377.773,A -85,B 0,C 180,E1 20884.315,E2 20884.315} C_VEL
LIN {X 0,Y 457.171,Z 374.752,A -85,B 0,C 180,E1 20883.888,E2 20883.888} C_VEL
LIN {X 0,Y 457.066,Z 374.115,A -85,B 0,C 180,E1 20883.386,E2 20883.386} C_VEL
LIN {X 0,Y 457.058,Z 374.109,A -85,B 0,C 180,E1 20879.624,E2 20879.624} C_VEL
LIN {X 0,Y 457.062,Z 374.11,A -85,B 0,C 180,E1 20875.861,E2 20875.861} C_VEL
LIN {X 0,Y 457.074,Z 374.105,A -85,B 0,C 180,E1 20872.206,E2 20872.206} C_VEL
LIN {X 0,Y 457.073,Z 374.113,A -85,B 0,C 180,E1 20868.518,E2 20868.518} C_VEL
LIN {X 0,Y 457.044,Z 374.114,A -85,B 0,C 180,E1 20864.911,E2 20864.911} C_VEL
LIN {X 0,Y 457.035,Z 374.118,A -85,B 0,C 180,E1 20861.241,E2 20861.241} C_VEL
LIN {X 0,Y 457.049,Z 374.118,A -85,B 0,C 180,E1 20857.627,E2 20857.627} C_VEL
LIN {X 0,Y 457.071,Z 374.113,A -85,B 0,C 180,E1 20854.04,E2 20854.04} C_VEL
LIN {X 0,Y 457.024,Z 374.109,A -85,B 0,C 180,E1 20850.512,E2 20850.512} C_VEL
LIN {X 0,Y 457.007,Z 374.122,A -85,B 0,C 180,E1 20846.842,E2 20846.842} C_VEL
LIN {X 0,Y 457.083,Z 374.368,A -85,B 0,C 180,E1 20845.559,E2 20845.559} C_VEL
LIN {X 0,Y 458.329,Z 377.63,A -85,B 0,C 180,E1 20844.836,E2 20844.836} C_VEL
LIN {X 0,Y 459.722,Z 379.455,A -85,B 0,C 180,E1 20844.347,E2 20844.347} C_VEL
LIN {X 0,Y 461.875,Z 383.583,A -85,B 0,C 180,E1 20843.465,E2 20843.465} C_VEL
LIN {X 0,Y 463.581,Z 386.653,A -85,B 0,C 180,E1 20842.966,E2 20842.966} C_VEL
LIN {X 0,Y 469.249,Z 394.232,A -85,B 0,C 180,E1 20841.797,E2 20841.797} C_VEL
LIN {X 0,Y 479.082,Z 408.565,A -85,B 0,C 180,E1 20839.921,E2 20839.921} C_VEL
LIN {X 0,Y 490.094,Z 425.986,A -85,B 0,C 180,E1 20837.998,E2 20837.998} C_VEL
LIN {X 0,Y 493.804,Z 432.317,A -85,B 0,C 180,E1 20837.382,E2 20837.382} C_VEL
LIN {X 0,Y 488.145,Z 635.554,A -85,B 0,C 180,E1 20833.825,E2 20833.825} C_VEL
LIN {X 0,Y 485.426,Z 739.56,A -85,B 0,C 180,E1 20832.027,E2 20832.027} C_VEL
LIN {X 0,Y 484.034,Z 762.614,A -85,B 0,C 180,E1 20831.441,E2 20831.441} C_VEL
LIN {X 0,Y 482.385,Z 784.666,A -85,B 0,C 180,E1 20830.685,E2 20830.685} C_VEL
LIN {X 0,Y 480.323,Z 806.22,A -85,B 0,C 180,E1 20829.724,E2 20829.724} C_VEL
LIN {X 0,Y 478.026,Z 827.714,A -85,B 0,C 180,E1 20828.561,E2 20828.561} C_VEL
LIN {X 0,Y 475.457,Z 848.915,A -85,B 0,C 180,E1 20827.155,E2 20827.155} C_VEL
LIN {X 0,Y 472.629,Z 870.834,A -85,B 0,C 180,E1 20825.429,E2 20825.429} C_VEL
LIN {X 0,Y 470.106,Z 889.346,A -85,B 0,C 180,E1 20823.721,E2 20823.721} C_VEL
LIN {X 0,Y 467.546,Z 907.755,A -85,B 0,C 180,E1 20821.743,E2 20821.743} C_VEL
LIN {X 0,Y 465.555,Z 921.609,A -85,B 0,C 180,E1 20820.029,E2 20820.029} C_VEL
LIN {X 0,Y 463.18,Z 938.272,A -85,B 0,C 180,E1 20817.656,E2 20817.656} C_VEL
LIN {X 0,Y 461.231,Z 952.717,A -85,B 0,C 180,E1 20815.284,E2 20815.284} C_VEL
LIN {X 0,Y 459.547,Z 966.188,A -85,B 0,C 180,E1 20812.704,E2 20812.704} C_VEL
LIN {X 0,Y 458.241,Z 978.242,A -85,B 0,C 180,E1 20810.036,E2 20810.036} C_VEL
